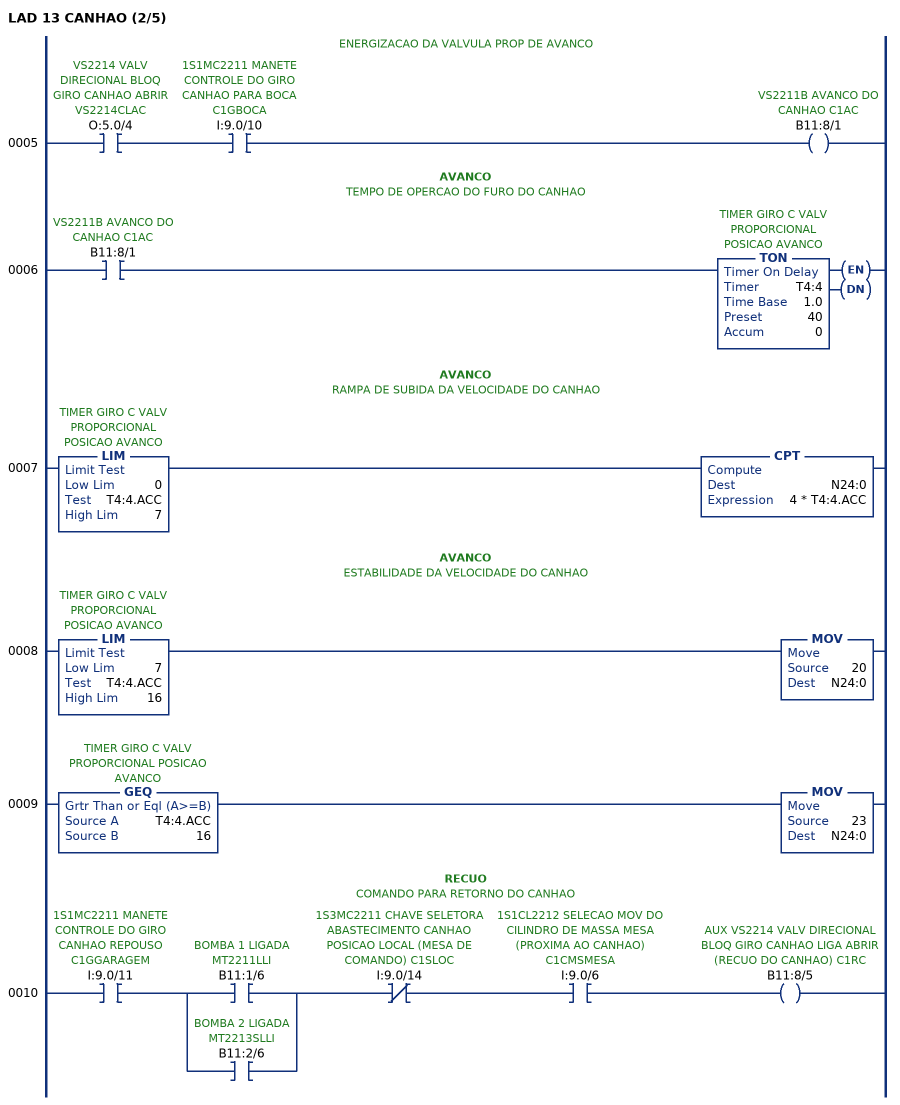
% Rung: 5 %
% ENERGIZACAO DA VALVULA PROP DE AVANCO %
SOR XIC O:5.0/4 XIC I:9.0/10 OTE B11:8/1 EOR
%   O:5.0/4  VS2214CLAC  "VS2214 VALV DIRECIONAL BLOQ GIRO CANHAO ABRIR" %
%   I:9.0/10  C1GBOCA  "1S1MC2211 MANETE CONTROLE DO GIRO CANHAO PARA BOCA" %
%   B11:8/1  C1AC  "VS2211B AVANCO DO CANHAO" %
% Rung: 6 %
% TITLE: AVANCO %
% TEMPO DE OPERCAO DO FURO DO CANHAO %
SOR XIC B11:8/1 TON T4:4 1.0 40 0 EOR
%   B11:8/1  C1AC  "VS2211B AVANCO DO CANHAO" %
%   T4:4  "TIMER GIRO C VALV PROPORCIONAL POSICAO AVANCO" %
% Rung: 7 %
% TITLE: AVANCO %
% RAMPA DE SUBIDA DA VELOCIDADE DO CANHAO %
SOR LIM 0 T4:4.ACC 7 CPT N24:0 " 4 * T4:4.ACC " EOR
%   T4:4  "TIMER GIRO C VALV PROPORCIONAL POSICAO AVANCO" %
% Rung: 8 %
% TITLE: AVANCO %
% ESTABILIDADE DA VELOCIDADE DO CANHAO %
SOR LIM 7 T4:4.ACC 16 MOV 20 N24:0 EOR
%   T4:4  "TIMER GIRO C VALV PROPORCIONAL POSICAO AVANCO" %
% Rung: 9 %
SOR GEQ T4:4.ACC 16 MOV 23 N24:0 EOR
%   T4:4  "TIMER GIRO C VALV PROPORCIONAL POSICAO AVANCO" %
% Rung: 10 %
% TITLE: RECUO %
% COMANDO PARA RETORNO DO CANHAO %
SOR XIC I:9.0/11 BST XIC B11:1/6 NXB XIC B11:2/6 BND XIO I:9.0/14 XIC I:9.0/6 OTE B11:8/5 EOR
%   I:9.0/11  C1GGARAGEM  "1S1MC2211 MANETE CONTROLE DO GIRO CANHAO REPOUSO" %
%   B11:1/6  MT2211LLI  "BOMBA 1 LIGADA" %
%   B11:2/6  MT2213SLLI  "BOMBA 2 LIGADA" %
%   I:9.0/14  C1SLOC  "1S3MC2211 CHAVE SELETORA ABASTECIMENTO CANHAO POSICAO LOCAL (MESA DE COMANDO)" %
%   I:9.0/6  C1CMSMESA  "1S1CL2212 SELECAO MOV DO CILINDRO DE MASSA MESA (PROXIMA AO CANHAO)" %
%   B11:8/5  C1RC  "AUX VS2214 VALV DIRECIONAL BLOQ GIRO CANHAO LIGA ABRIR (RECUO DO CANHAO)" %

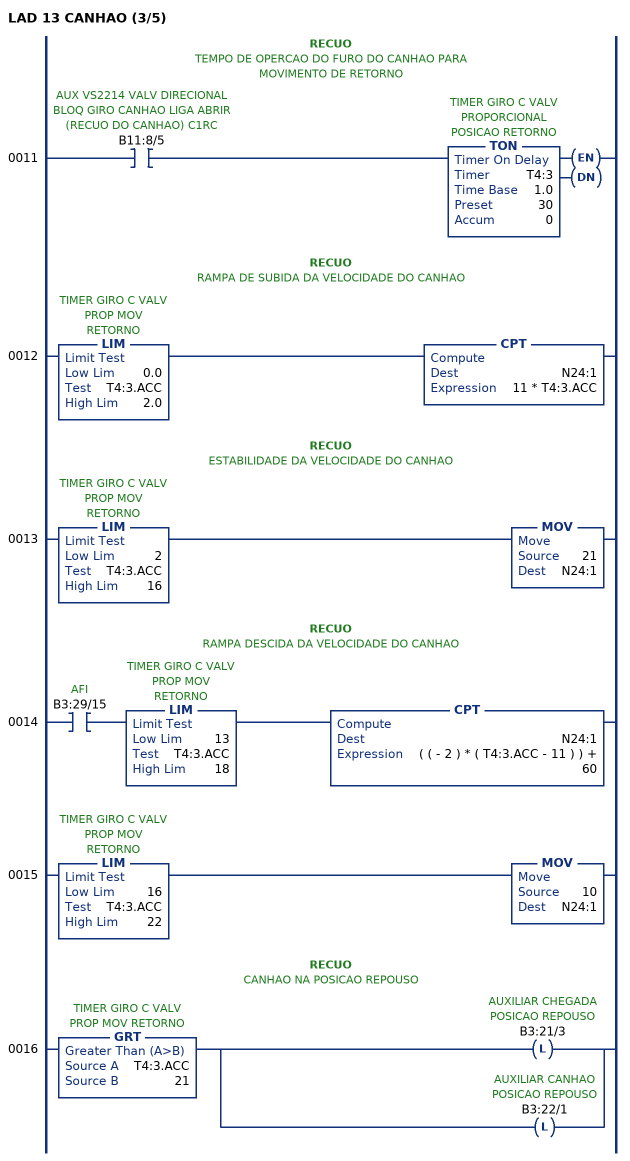
% Rung: 11 %
% TITLE: RECUO %
% TEMPO DE OPERCAO DO FURO DO CANHAO PARA
%  MOVIMENTO DE RETORNO %
SOR XIC B11:8/5 TON T4:3 1.0 30 0 EOR
%   B11:8/5  C1RC  "AUX VS2214 VALV DIRECIONAL BLOQ GIRO CANHAO LIGA ABRIR (RECUO DO CANHAO)" %
%   T4:3  "TIMER GIRO C VALV PROPORCIONAL POSICAO RETORNO" %
% Rung: 12 %
% TITLE: RECUO %
% RAMPA DE SUBIDA DA VELOCIDADE DO CANHAO %
SOR LIM 0.0 T4:3.ACC 2.0 CPT N24:1 " 11 * T4:3.ACC " EOR
%   T4:3.ACC  "TIMER GIRO C VALV PROP MOV RETORNO" %
% Rung: 13 %
% TITLE: RECUO %
% ESTABILIDADE DA VELOCIDADE DO CANHAO %
SOR LIM 2 T4:3.ACC 16 MOV 21 N24:1 EOR
%   T4:3.ACC  "TIMER GIRO C VALV PROP MOV RETORNO" %
% Rung: 14 %
% TITLE: RECUO %
% RAMPA DESCIDA DA VELOCIDADE DO CANHAO %
SOR XIC B3:29/15 LIM 13 T4:3.ACC 18 CPT N24:1 " ( ( - 2 ) * ( T4:3.ACC - 11 ) ) + 60 " EOR
%   B3:29/15  AFI %
%   T4:3.ACC  "TIMER GIRO C VALV PROP MOV RETORNO" %
% Rung: 15 %
SOR LIM 16 T4:3.ACC 22 MOV 10 N24:1 EOR
%   T4:3.ACC  "TIMER GIRO C VALV PROP MOV RETORNO" %
% Rung: 16 %
% TITLE: RECUO %
% CANHAO NA POSICAO REPOUSO %
SOR GRT T4:3.ACC 21 BST OTL B3:21/3 NXB OTL B3:22/1 BND EOR
%   T4:3.ACC  "TIMER GIRO C VALV PROP MOV RETORNO" %
%   B3:21/3  "AUXILIAR CHEGADA POSICAO REPOUSO" %
%   B3:22/1  "AUXILIAR CANHAO POSICAO REPOUSO" %

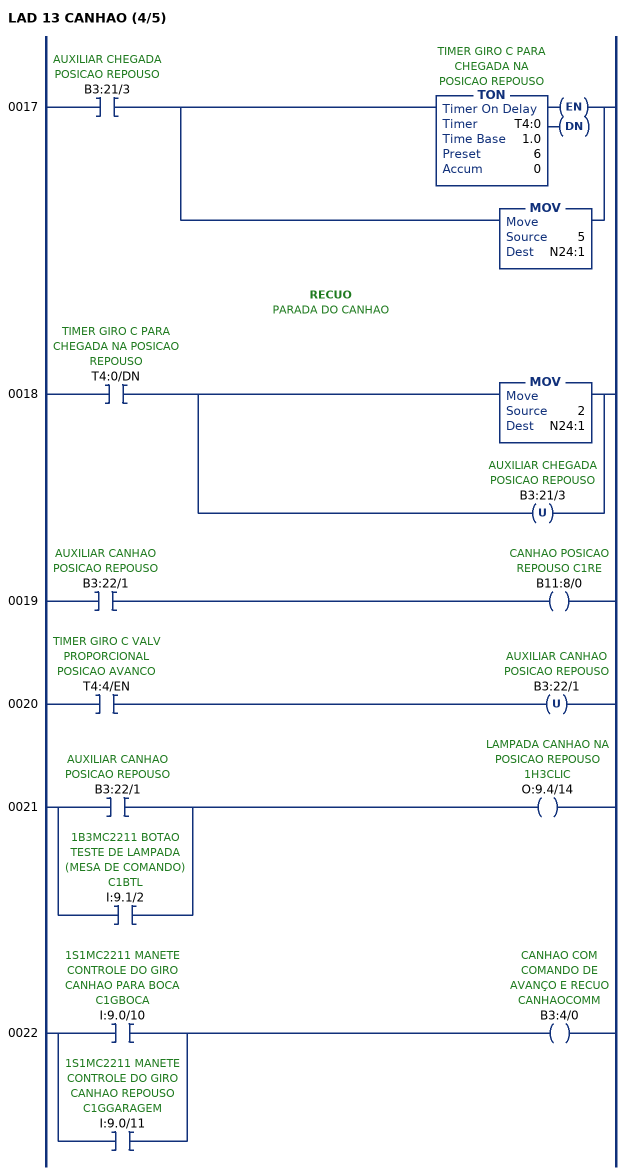
% Rung: 17 %
SOR XIC B3:21/3 BST TON T4:0 1.0 6 0 NXB MOV 5 N24:1 BND EOR
%   B3:21/3  "AUXILIAR CHEGADA POSICAO REPOUSO" %
%   T4:0  "TIMER GIRO C PARA CHEGADA NA POSICAO REPOUSO" %
% Rung: 18 %
% TITLE: RECUO %
% PARADA DO CANHAO %
SOR XIC T4:0/DN BST MOV 2 N24:1 NXB OTU B3:21/3 BND EOR
%   T4:0  "TIMER GIRO C PARA CHEGADA NA POSICAO REPOUSO" %
%   B3:21/3  "AUXILIAR CHEGADA POSICAO REPOUSO" %
% Rung: 19 %
SOR XIC B3:22/1 OTE B11:8/0 EOR
%   B3:22/1  "AUXILIAR CANHAO POSICAO REPOUSO" %
%   B11:8/0  C1RE  "CANHAO POSICAO REPOUSO" %
% Rung: 20 %
SOR XIC T4:4/EN OTU B3:22/1 EOR
%   T4:4  "TIMER GIRO C VALV PROPORCIONAL POSICAO AVANCO" %
%   B3:22/1  "AUXILIAR CANHAO POSICAO REPOUSO" %
% Rung: 21 %
SOR BST XIC B3:22/1 NXB XIC I:9.1/2 BND OTE O:9.4/14 EOR
%   B3:22/1  "AUXILIAR CANHAO POSICAO REPOUSO" %
%   I:9.1/2  C1BTL  "1B3MC2211 BOTAO TESTE DE LAMPADA (MESA DE COMANDO)" %
%   O:9.4/14  1H3CLIC  "LAMPADA CANHAO NA POSICAO REPOUSO" %
% Rung: 22 %
SOR BST XIC I:9.0/10 NXB XIC I:9.0/11 BND OTE B3:4/0 EOR
%   I:9.0/10  C1GBOCA  "1S1MC2211 MANETE CONTROLE DO GIRO CANHAO PARA BOCA" %
%   I:9.0/11  C1GGARAGEM  "1S1MC2211 MANETE CONTROLE DO GIRO CANHAO REPOUSO" %
%   B3:4/0  CANHAOCOMM  "CANHAO COM COMANDO DE AVANÇO E RECUO" %

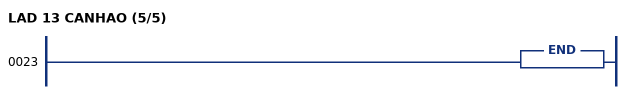
% Rung: 23 %
SOR END EOR

LADDER 14 "INJECAO M"
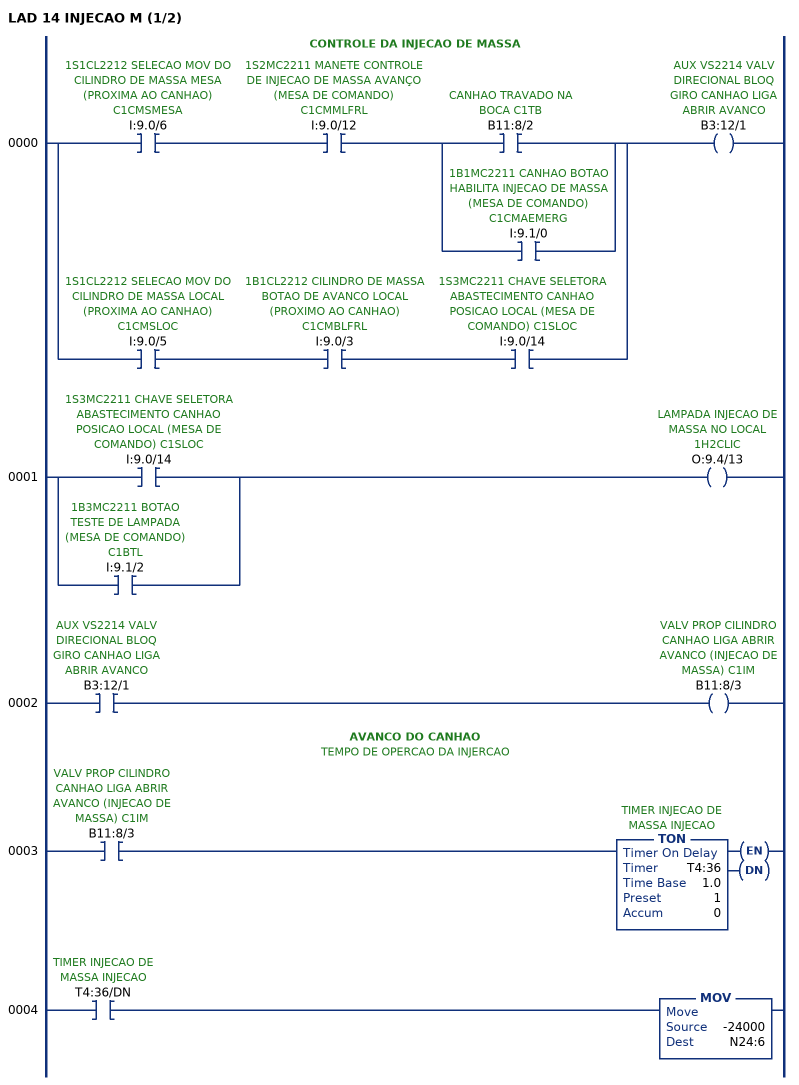
% Rung: 0 %
% TITLE: CONTROLE DA INJECAO DE MASSA %
SOR BST XIC I:9.0/6 XIC I:9.0/12 BST XIC B11:8/2 NXB XIC I:9.1/0 BND NXB XIC I:9.0/5 XIC I:9.0/3 XIC I:9.0/14 BND OTE B3:12/1 EOR
%   I:9.0/6  C1CMSMESA  "1S1CL2212 SELECAO MOV DO CILINDRO DE MASSA MESA (PROXIMA AO CANHAO)" %
%   I:9.0/12  C1CMMLFRL  "1S2MC2211 MANETE CONTROLE DE INJECAO DE MASSA AVANÇO (MESA DE COMANDO)" %
%   B11:8/2  C1TB  "CANHAO TRAVADO NA BOCA" %
%   I:9.1/0  C1CMAEMERG  "1B1MC2211 CANHAO BOTAO HABILITA INJECAO DE MASSA (MESA DE COMANDO)" %
%   I:9.0/5  C1CMSLOC  "1S1CL2212 SELECAO MOV DO CILINDRO DE MASSA LOCAL (PROXIMA AO CANHAO)" %
%   I:9.0/3  C1CMBLFRL  "1B1CL2212 CILINDRO DE MASSA BOTAO DE AVANCO LOCAL (PROXIMO AO CANHAO)" %
%   I:9.0/14  C1SLOC  "1S3MC2211 CHAVE SELETORA ABASTECIMENTO CANHAO POSICAO LOCAL (MESA DE COMANDO)" %
%   B3:12/1  "AUX VS2214 VALV DIRECIONAL BLOQ GIRO CANHAO LIGA ABRIR AVANCO" %
% Rung: 1 %
SOR BST XIC I:9.0/14 NXB XIC I:9.1/2 BND OTE O:9.4/13 EOR
%   I:9.0/14  C1SLOC  "1S3MC2211 CHAVE SELETORA ABASTECIMENTO CANHAO POSICAO LOCAL (MESA DE COMANDO)" %
%   I:9.1/2  C1BTL  "1B3MC2211 BOTAO TESTE DE LAMPADA (MESA DE COMANDO)" %
%   O:9.4/13  1H2CLIC  "LAMPADA INJECAO DE MASSA NO LOCAL" %
% Rung: 2 %
SOR XIC B3:12/1 OTE B11:8/3 EOR
%   B3:12/1  "AUX VS2214 VALV DIRECIONAL BLOQ GIRO CANHAO LIGA ABRIR AVANCO" %
%   B11:8/3  C1IM  "VALV PROP CILINDRO CANHAO LIGA ABRIR AVANCO (INJECAO DE MASSA)" %
% Rung: 3 %
% TITLE: AVANCO DO CANHAO %
% TEMPO DE OPERCAO DA INJERCAO %
SOR XIC B11:8/3 TON T4:36 1.0 1 0 EOR
%   B11:8/3  C1IM  "VALV PROP CILINDRO CANHAO LIGA ABRIR AVANCO (INJECAO DE MASSA)" %
%   T4:36  "TIMER INJECAO DE MASSA INJECAO" %
% Rung: 4 %
SOR XIC T4:36/DN MOV -24000 N24:6 EOR
%   T4:36  "TIMER INJECAO DE MASSA INJECAO" %

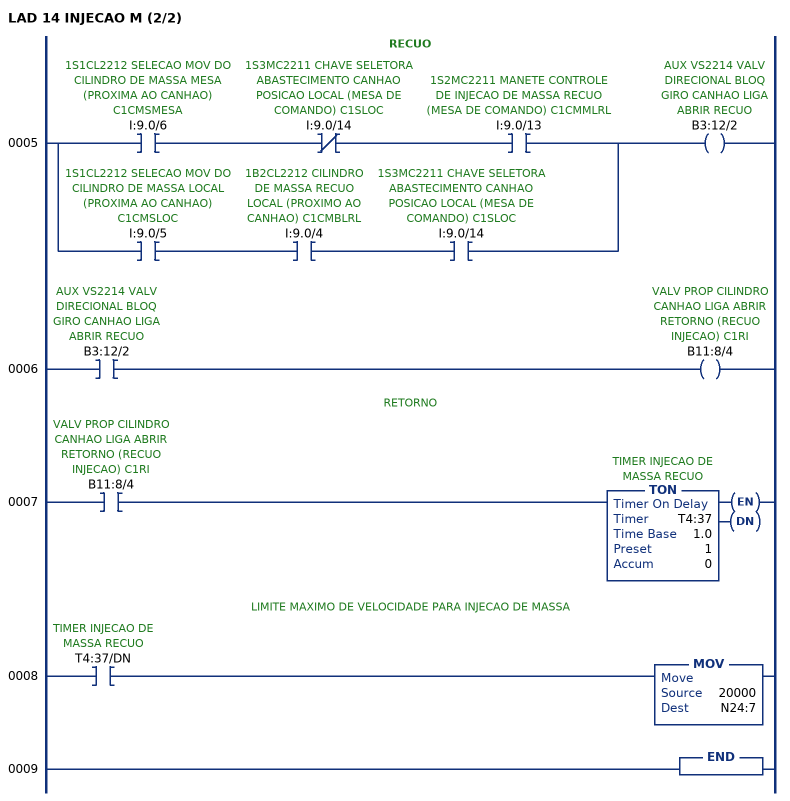
% Rung: 5 %
% TITLE: RECUO %
SOR BST XIC I:9.0/6 XIO I:9.0/14 XIC I:9.0/13 NXB XIC I:9.0/5 XIC I:9.0/4 XIC I:9.0/14 BND OTE B3:12/2 EOR
%   I:9.0/6  C1CMSMESA  "1S1CL2212 SELECAO MOV DO CILINDRO DE MASSA MESA (PROXIMA AO CANHAO)" %
%   I:9.0/14  C1SLOC  "1S3MC2211 CHAVE SELETORA ABASTECIMENTO CANHAO POSICAO LOCAL (MESA DE COMANDO)" %
%   I:9.0/13  C1CMMLRL  "1S2MC2211 MANETE CONTROLE DE INJECAO DE MASSA RECUO (MESA DE COMANDO)" %
%   I:9.0/5  C1CMSLOC  "1S1CL2212 SELECAO MOV DO CILINDRO DE MASSA LOCAL (PROXIMA AO CANHAO)" %
%   I:9.0/4  C1CMBLRL  "1B2CL2212 CILINDRO DE MASSA RECUO LOCAL (PROXIMO AO CANHAO)" %
%   B3:12/2  "AUX VS2214 VALV DIRECIONAL BLOQ GIRO CANHAO LIGA ABRIR RECUO" %
% Rung: 6 %
SOR XIC B3:12/2 OTE B11:8/4 EOR
%   B3:12/2  "AUX VS2214 VALV DIRECIONAL BLOQ GIRO CANHAO LIGA ABRIR RECUO" %
%   B11:8/4  C1RI  "VALV PROP CILINDRO CANHAO LIGA ABRIR RETORNO (RECUO INJECAO)" %
% Rung: 7 %
% RETORNO %
SOR XIC B11:8/4 TON T4:37 1.0 1 0 EOR
%   B11:8/4  C1RI  "VALV PROP CILINDRO CANHAO LIGA ABRIR RETORNO (RECUO INJECAO)" %
%   T4:37  "TIMER INJECAO DE MASSA RECUO" %
% Rung: 8 %
% LIMITE MAXIMO DE VELOCIDADE PARA INJECAO DE MASSA %
SOR XIC T4:37/DN MOV 20000 N24:7 EOR
%   T4:37  "TIMER INJECAO DE MASSA RECUO" %
% Rung: 9 %
SOR END EOR

LADDER 15 "PERFURAT"
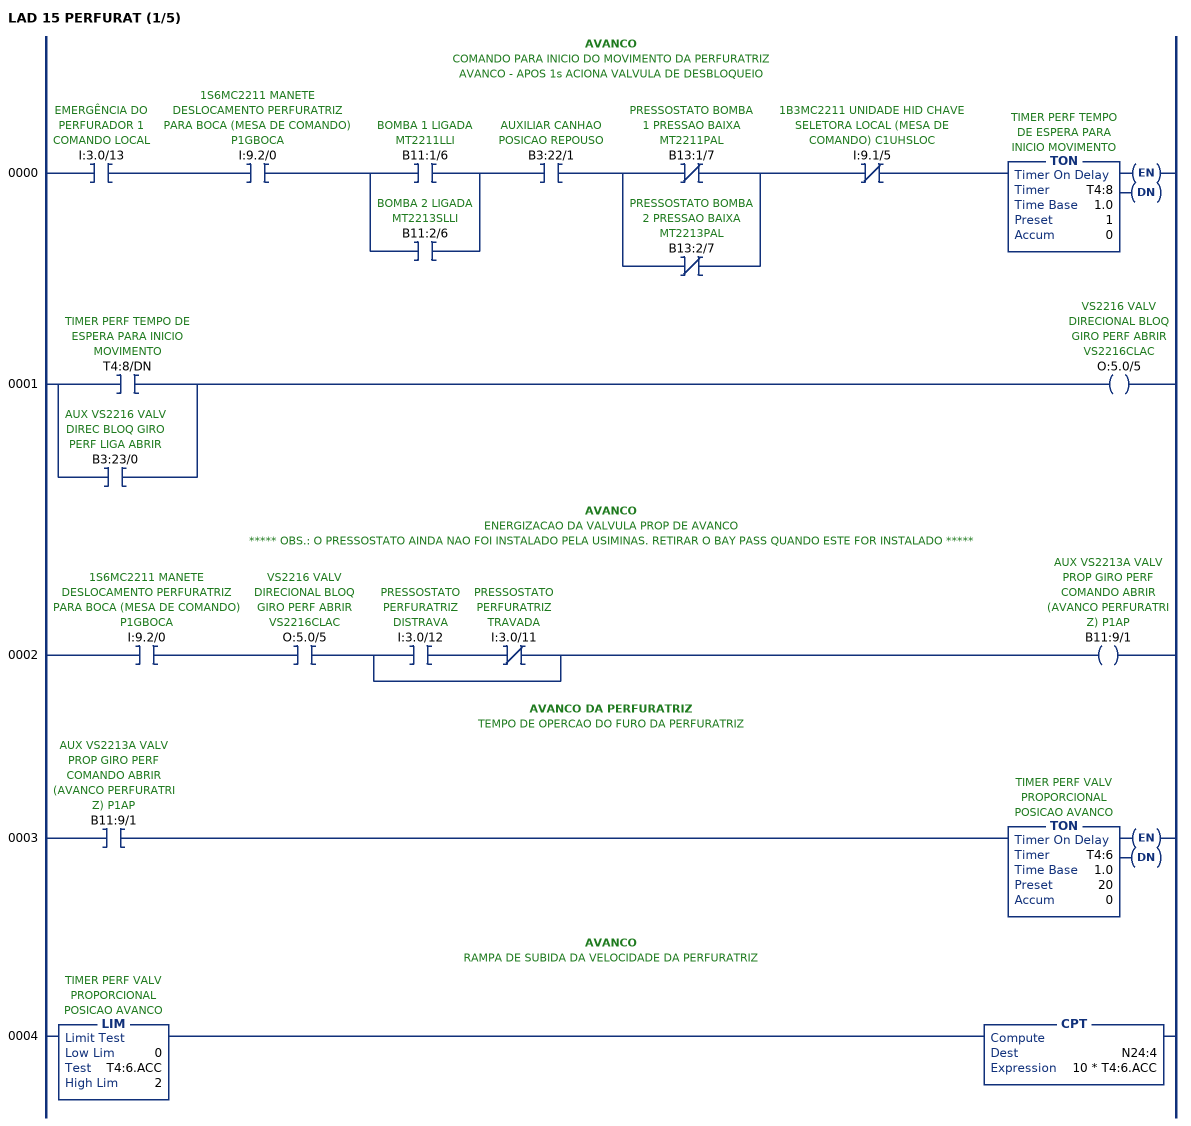
% Rung: 0 %
% TITLE: AVANCO %
% COMANDO PARA INICIO DO MOVIMENTO DA PERFURATRIZ
% AVANCO - APOS 1s ACIONA VALVULA DE DESBLOQUEIO %
SOR XIC I:3.0/13 XIC I:9.2/0 BST XIC B11:1/6 NXB XIC B11:2/6 BND XIC B3:22/1 BST XIO B13:1/7 NXB XIO B13:2/7 BND XIO I:9.1/5 TON T4:8 1.0 1 0 EOR
%   I:3.0/13  "EMERGÊNCIA DO PERFURADOR 1 COMANDO LOCAL" %
%   I:9.2/0  P1GBOCA  "1S6MC2211 MANETE DESLOCAMENTO PERFURATRIZ PARA BOCA (MESA DE COMANDO)" %
%   B11:1/6  MT2211LLI  "BOMBA 1 LIGADA" %
%   B11:2/6  MT2213SLLI  "BOMBA 2 LIGADA" %
%   B3:22/1  "AUXILIAR CANHAO POSICAO REPOUSO" %
%   B13:1/7  MT2211PAL  "PRESSOSTATO BOMBA 1 PRESSAO BAIXA" %
%   B13:2/7  MT2213PAL  "PRESSOSTATO BOMBA 2 PRESSAO BAIXA" %
%   I:9.1/5  C1UHSLOC  "1B3MC2211 UNIDADE HID CHAVE SELETORA LOCAL (MESA DE COMANDO)" %
%   T4:8  "TIMER PERF TEMPO DE ESPERA PARA INICIO MOVIMENTO" %
% Rung: 1 %
SOR BST XIC T4:8/DN NXB XIC B3:23/0 BND OTE O:5.0/5 EOR
%   T4:8  "TIMER PERF TEMPO DE ESPERA PARA INICIO MOVIMENTO" %
%   B3:23/0  "AUX VS2216 VALV DIREC BLOQ GIRO PERF LIGA ABRIR" %
%   O:5.0/5  VS2216CLAC  "VS2216 VALV DIRECIONAL BLOQ GIRO PERF ABRIR" %
% Rung: 2 %
% TITLE: AVANCO %
% ENERGIZACAO DA VALVULA PROP DE AVANCO
% ***** OBS.: O PRESSOSTATO AINDA NAO FOI INSTALADO PELA USIMINAS. RETIRAR O BAY PASS QUANDO ESTE FOR INSTALADO ***** %
SOR XIC I:9.2/0 XIC O:5.0/5 BST XIC I:3.0/12 XIO I:3.0/11 NXB BND OTE B11:9/1 EOR
%   I:9.2/0  P1GBOCA  "1S6MC2211 MANETE DESLOCAMENTO PERFURATRIZ PARA BOCA (MESA DE COMANDO)" %
%   O:5.0/5  VS2216CLAC  "VS2216 VALV DIRECIONAL BLOQ GIRO PERF ABRIR" %
%   I:3.0/12  "PRESSOSTATO PERFURATRIZ DISTRAVA" %
%   I:3.0/11  "PRESSOSTATO PERFURATRIZ TRAVADA" %
%   B11:9/1  P1AP  "AUX VS2213A VALV PROP GIRO PERF COMANDO ABRIR (AVANCO PERFURATRIZ)" %
% Rung: 3 %
% TITLE: AVANCO DA PERFURATRIZ %
% TEMPO DE OPERCAO DO FURO DA PERFURATRIZ %
SOR XIC B11:9/1 TON T4:6 1.0 20 0 EOR
%   B11:9/1  P1AP  "AUX VS2213A VALV PROP GIRO PERF COMANDO ABRIR (AVANCO PERFURATRIZ)" %
%   T4:6  "TIMER PERF VALV PROPORCIONAL POSICAO AVANCO" %
% Rung: 4 %
% TITLE: AVANCO %
% RAMPA DE SUBIDA DA VELOCIDADE DA PERFURATRIZ %
SOR LIM 0 T4:6.ACC 2 CPT N24:4 " 10 * T4:6.ACC " EOR
%   T4:6  "TIMER PERF VALV PROPORCIONAL POSICAO AVANCO" %

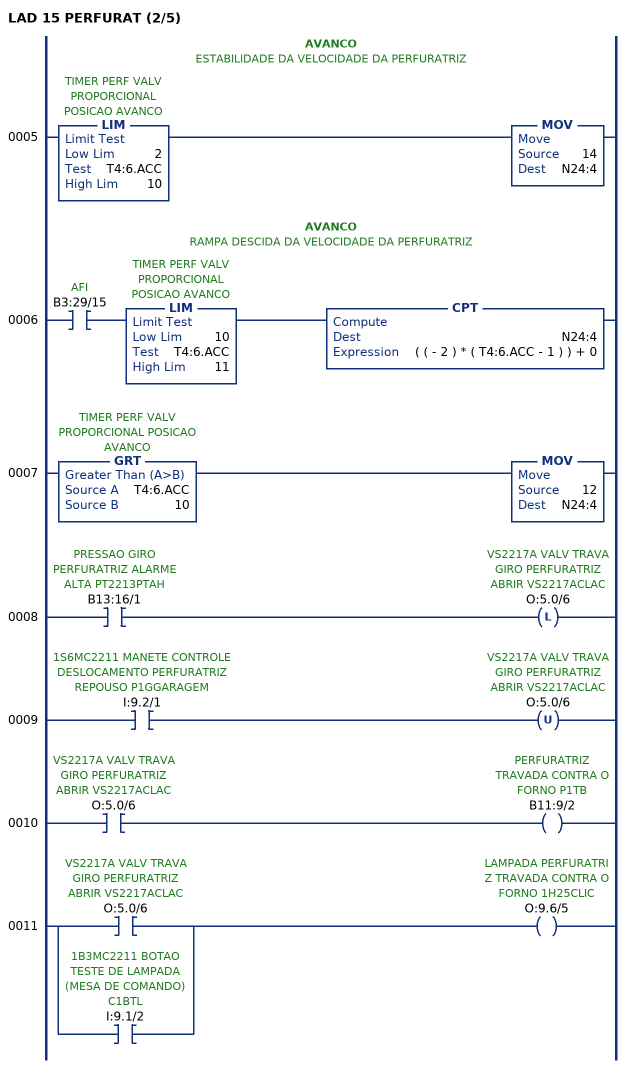
% Rung: 5 %
% TITLE: AVANCO %
% ESTABILIDADE DA VELOCIDADE DA PERFURATRIZ %
SOR LIM 2 T4:6.ACC 10 MOV 14 N24:4 EOR
%   T4:6  "TIMER PERF VALV PROPORCIONAL POSICAO AVANCO" %
% Rung: 6 %
% TITLE: AVANCO %
% RAMPA DESCIDA DA VELOCIDADE DA PERFURATRIZ %
SOR XIC B3:29/15 LIM 10 T4:6.ACC 11 CPT N24:4 " ( ( - 2 ) * ( T4:6.ACC - 1 ) ) + 0 " EOR
%   B3:29/15  AFI %
%   T4:6  "TIMER PERF VALV PROPORCIONAL POSICAO AVANCO" %
% Rung: 7 %
SOR GRT T4:6.ACC 10 MOV 12 N24:4 EOR
%   T4:6  "TIMER PERF VALV PROPORCIONAL POSICAO AVANCO" %
% Rung: 8 %
SOR XIC B13:16/1 OTL O:5.0/6 EOR
%   B13:16/1  PT2213PTAH  "PRESSAO GIRO PERFURATRIZ ALARME ALTA" %
%   O:5.0/6  VS2217ACLAC  "VS2217A VALV TRAVA GIRO PERFURATRIZ ABRIR" %
% Rung: 9 %
SOR XIC I:9.2/1 OTU O:5.0/6 EOR
%   I:9.2/1  P1GGARAGEM  "1S6MC2211 MANETE CONTROLE DESLOCAMENTO PERFURATRIZ REPOUSO" %
%   O:5.0/6  VS2217ACLAC  "VS2217A VALV TRAVA GIRO PERFURATRIZ ABRIR" %
% Rung: 10 %
SOR XIC O:5.0/6 OTE B11:9/2 EOR
%   O:5.0/6  VS2217ACLAC  "VS2217A VALV TRAVA GIRO PERFURATRIZ ABRIR" %
%   B11:9/2  P1TB  "PERFURATRIZ TRAVADA CONTRA O FORNO" %
% Rung: 11 %
SOR BST XIC O:5.0/6 NXB XIC I:9.1/2 BND OTE O:9.6/5 EOR
%   O:5.0/6  VS2217ACLAC  "VS2217A VALV TRAVA GIRO PERFURATRIZ ABRIR" %
%   I:9.1/2  C1BTL  "1B3MC2211 BOTAO TESTE DE LAMPADA (MESA DE COMANDO)" %
%   O:9.6/5  1H25CLIC  "LAMPADA PERFURATRIZ TRAVADA CONTRA O FORNO" %

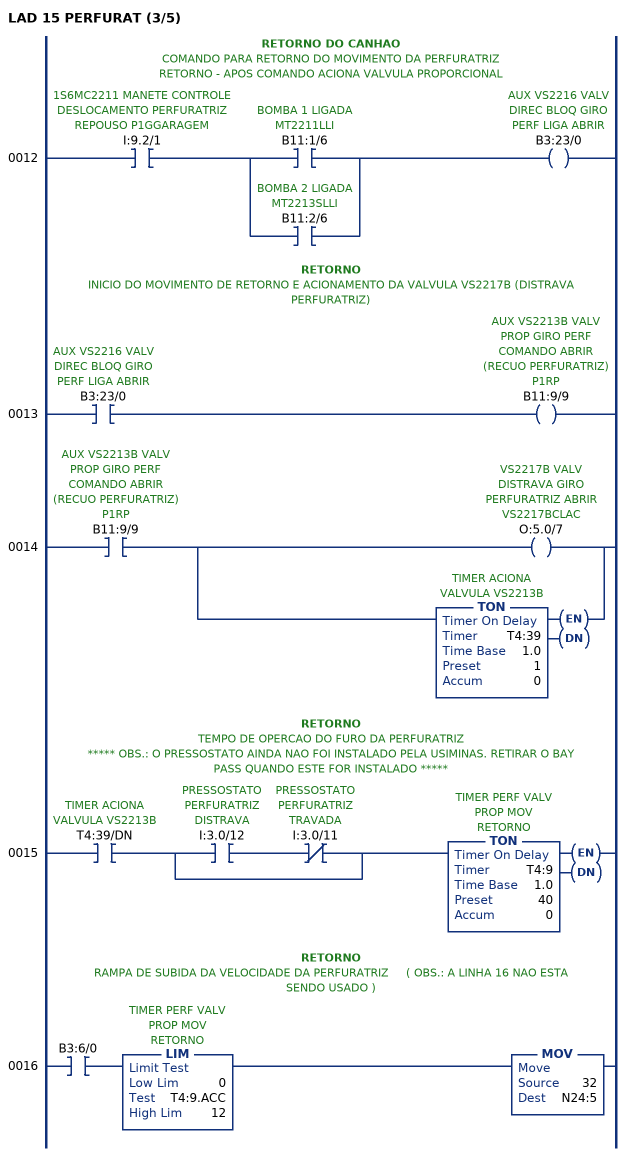
% Rung: 12 %
% TITLE: RETORNO DO CANHAO %
% COMANDO PARA RETORNO DO MOVIMENTO DA PERFURATRIZ
% RETORNO - APOS COMANDO ACIONA VALVULA PROPORCIONAL %
SOR XIC I:9.2/1 BST XIC B11:1/6 NXB XIC B11:2/6 BND OTE B3:23/0 EOR
%   I:9.2/1  P1GGARAGEM  "1S6MC2211 MANETE CONTROLE DESLOCAMENTO PERFURATRIZ REPOUSO" %
%   B11:1/6  MT2211LLI  "BOMBA 1 LIGADA" %
%   B11:2/6  MT2213SLLI  "BOMBA 2 LIGADA" %
%   B3:23/0  "AUX VS2216 VALV DIREC BLOQ GIRO PERF LIGA ABRIR" %
% Rung: 13 %
% TITLE: RETORNO %
% INICIO DO MOVIMENTO DE RETORNO E ACIONAMENTO DA VALVULA VS2217B (DISTRAVA PERFURATRIZ) %
SOR XIC B3:23/0 OTE B11:9/9 EOR
%   B3:23/0  "AUX VS2216 VALV DIREC BLOQ GIRO PERF LIGA ABRIR" %
%   B11:9/9  P1RP  "AUX VS2213B VALV PROP GIRO PERF COMANDO ABRIR (RECUO PERFURATRIZ)" %
% Rung: 14 %
SOR XIC B11:9/9 BST OTE O:5.0/7 NXB TON T4:39 1.0 1 0 BND EOR
%   B11:9/9  P1RP  "AUX VS2213B VALV PROP GIRO PERF COMANDO ABRIR (RECUO PERFURATRIZ)" %
%   O:5.0/7  VS2217BCLAC  "VS2217B VALV DISTRAVA GIRO PERFURATRIZ ABRIR" %
%   T4:39  "TIMER ACIONA VALVULA VS2213B" %
% Rung: 15 %
% TITLE: RETORNO %
% TEMPO DE OPERCAO DO FURO DA PERFURATRIZ
% ***** OBS.: O PRESSOSTATO AINDA NAO FOI INSTALADO PELA USIMINAS. RETIRAR O BAY PASS QUANDO ESTE FOR INSTALADO ***** %
SOR XIC T4:39/DN BST XIC I:3.0/12 XIO I:3.0/11 NXB BND TON T4:9 1.0 40 0 EOR
%   T4:39  "TIMER ACIONA VALVULA VS2213B" %
%   I:3.0/12  "PRESSOSTATO PERFURATRIZ DISTRAVA" %
%   I:3.0/11  "PRESSOSTATO PERFURATRIZ TRAVADA" %
%   T4:9  "TIMER PERF VALV PROP MOV RETORNO" %
% Rung: 16 %
% TITLE: RETORNO %
% RAMPA DE SUBIDA DA VELOCIDADE DA PERFURATRIZ     ( OBS.: A LINHA 16 NAO ESTA SENDO USADO ) %
SOR XIC B3:6/0 LIM 0 T4:9.ACC 12 MOV 32 N24:5 EOR
%   T4:9  "TIMER PERF VALV PROP MOV RETORNO" %

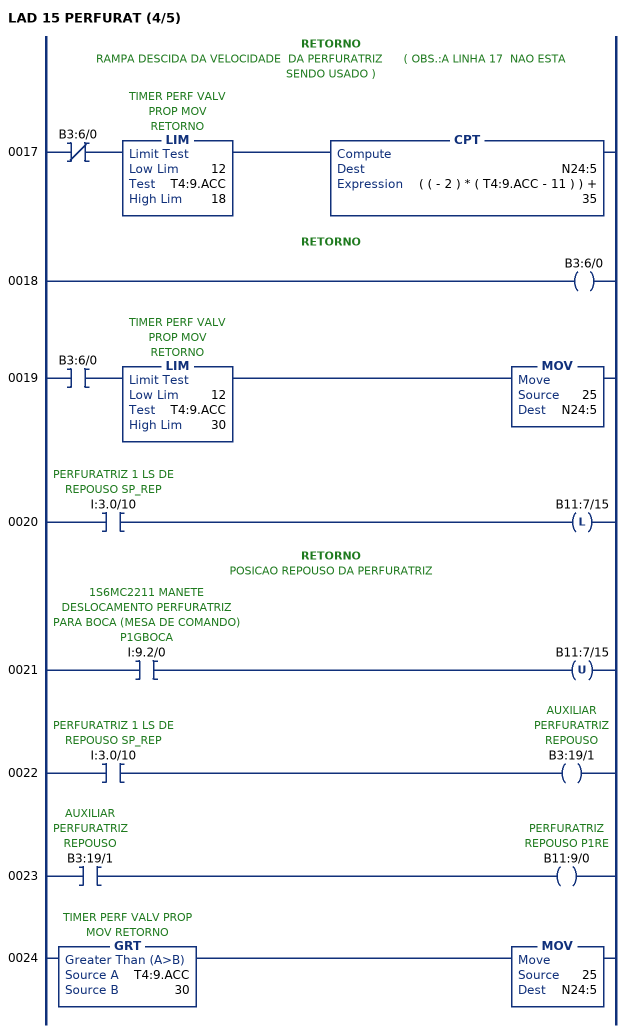
% Rung: 17 %
% TITLE: RETORNO %
% RAMPA DESCIDA DA VELOCIDADE  DA PERFURATRIZ      ( OBS.:A LINHA 17  NAO ESTA SENDO USADO ) %
SOR XIO B3:6/0 LIM 12 T4:9.ACC 18 CPT N24:5 " ( ( - 2 ) * ( T4:9.ACC - 11 ) ) + 35 " EOR
%   T4:9  "TIMER PERF VALV PROP MOV RETORNO" %
% Rung: 18 %
% TITLE: RETORNO %
SOR OTE B3:6/0 EOR
% Rung: 19 %
SOR XIC B3:6/0 LIM 12 T4:9.ACC 30 MOV 25 N24:5 EOR
%   T4:9  "TIMER PERF VALV PROP MOV RETORNO" %
% Rung: 20 %
SOR XIC I:3.0/10 OTL B11:7/15 EOR
%   I:3.0/10  SP_REP  "PERFURATRIZ 1 LS DE REPOUSO" %
% Rung: 21 %
% TITLE: RETORNO %
% POSICAO REPOUSO DA PERFURATRIZ %
SOR XIC I:9.2/0 OTU B11:7/15 EOR
%   I:9.2/0  P1GBOCA  "1S6MC2211 MANETE DESLOCAMENTO PERFURATRIZ PARA BOCA (MESA DE COMANDO)" %
% Rung: 22 %
SOR XIC I:3.0/10 OTE B3:19/1 EOR
%   I:3.0/10  SP_REP  "PERFURATRIZ 1 LS DE REPOUSO" %
%   B3:19/1  "AUXILIAR PERFURATRIZ REPOUSO" %
% Rung: 23 %
SOR XIC B3:19/1 OTE B11:9/0 EOR
%   B3:19/1  "AUXILIAR PERFURATRIZ REPOUSO" %
%   B11:9/0  P1RE  "PERFURATRIZ REPOUSO" %
% Rung: 24 %
SOR GRT T4:9.ACC 30 MOV 25 N24:5 EOR
%   T4:9  "TIMER PERF VALV PROP MOV RETORNO" %

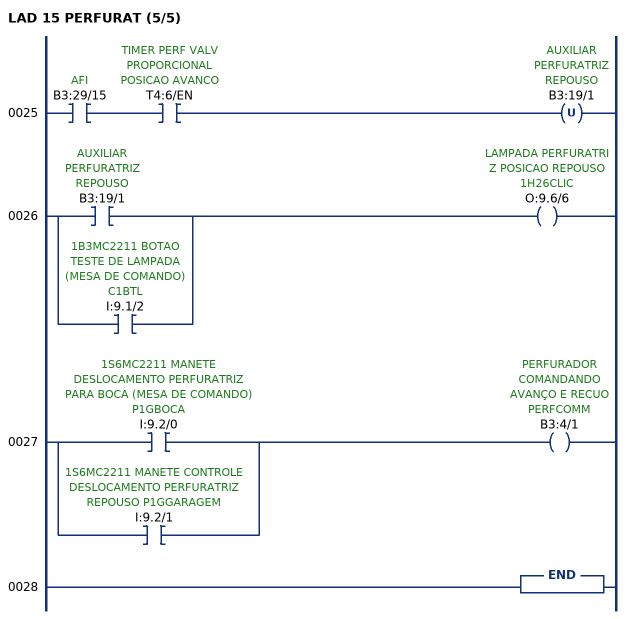
% Rung: 25 %
SOR XIC B3:29/15 XIC T4:6/EN OTU B3:19/1 EOR
%   B3:29/15  AFI %
%   T4:6  "TIMER PERF VALV PROPORCIONAL POSICAO AVANCO" %
%   B3:19/1  "AUXILIAR PERFURATRIZ REPOUSO" %
% Rung: 26 %
SOR BST XIC B3:19/1 NXB XIC I:9.1/2 BND OTE O:9.6/6 EOR
%   B3:19/1  "AUXILIAR PERFURATRIZ REPOUSO" %
%   I:9.1/2  C1BTL  "1B3MC2211 BOTAO TESTE DE LAMPADA (MESA DE COMANDO)" %
%   O:9.6/6  1H26CLIC  "LAMPADA PERFURATRIZ POSICAO REPOUSO" %
% Rung: 27 %
SOR BST XIC I:9.2/0 NXB XIC I:9.2/1 BND OTE B3:4/1 EOR
%   I:9.2/0  P1GBOCA  "1S6MC2211 MANETE DESLOCAMENTO PERFURATRIZ PARA BOCA (MESA DE COMANDO)" %
%   I:9.2/1  P1GGARAGEM  "1S6MC2211 MANETE CONTROLE DESLOCAMENTO PERFURATRIZ REPOUSO" %
%   B3:4/1  PERFCOMM  "PERFURADOR COMANDANDO AVANÇO E RECUO" %
% Rung: 28 %
SOR END EOR

LADDER 16 "MARTELETE"
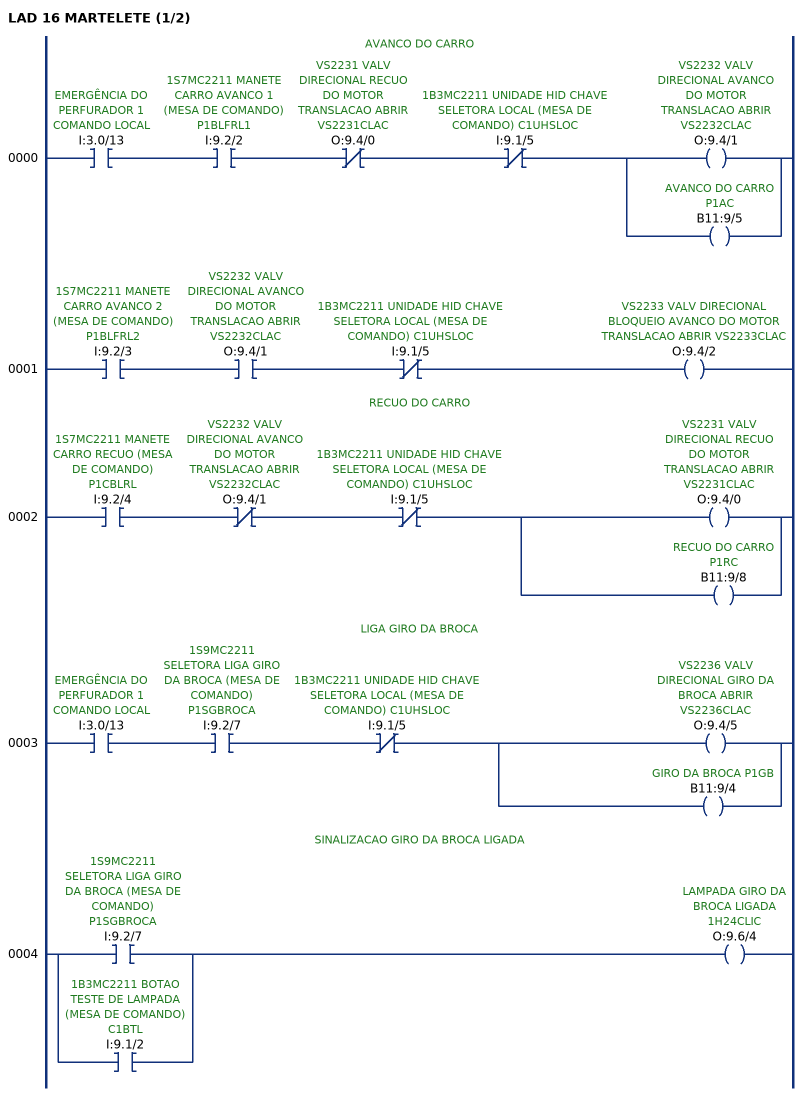
% Rung: 0 %
% AVANCO DO CARRO %
SOR XIC I:3.0/13 XIC I:9.2/2 XIO O:9.4/0 XIO I:9.1/5 BST OTE O:9.4/1 NXB OTE B11:9/5 BND EOR
%   I:3.0/13  "EMERGÊNCIA DO PERFURADOR 1 COMANDO LOCAL" %
%   I:9.2/2  P1BLFRL1  "1S7MC2211 MANETE CARRO AVANCO 1 (MESA DE COMANDO)" %
%   O:9.4/0  VS2231CLAC  "VS2231 VALV DIRECIONAL RECUO DO MOTOR TRANSLACAO ABRIR" %
%   I:9.1/5  C1UHSLOC  "1B3MC2211 UNIDADE HID CHAVE SELETORA LOCAL (MESA DE COMANDO)" %
%   O:9.4/1  VS2232CLAC  "VS2232 VALV DIRECIONAL AVANCO DO MOTOR TRANSLACAO ABRIR" %
%   B11:9/5  P1AC  "AVANCO DO CARRO" %
% Rung: 1 %
SOR XIC I:9.2/3 XIC O:9.4/1 XIO I:9.1/5 OTE O:9.4/2 EOR
%   I:9.2/3  P1BLFRL2  "1S7MC2211 MANETE CARRO AVANCO 2 (MESA DE COMANDO)" %
%   O:9.4/1  VS2232CLAC  "VS2232 VALV DIRECIONAL AVANCO DO MOTOR TRANSLACAO ABRIR" %
%   I:9.1/5  C1UHSLOC  "1B3MC2211 UNIDADE HID CHAVE SELETORA LOCAL (MESA DE COMANDO)" %
%   O:9.4/2  VS2233CLAC  "VS2233 VALV DIRECIONAL BLOQUEIO AVANCO DO MOTOR TRANSLACAO ABRIR" %
% Rung: 2 %
% RECUO DO CARRO %
SOR XIC I:9.2/4 XIO O:9.4/1 XIO I:9.1/5 BST OTE O:9.4/0 NXB OTE B11:9/8 BND EOR
%   I:9.2/4  P1CBLRL  "1S7MC2211 MANETE CARRO RECUO (MESA DE COMANDO)" %
%   O:9.4/1  VS2232CLAC  "VS2232 VALV DIRECIONAL AVANCO DO MOTOR TRANSLACAO ABRIR" %
%   I:9.1/5  C1UHSLOC  "1B3MC2211 UNIDADE HID CHAVE SELETORA LOCAL (MESA DE COMANDO)" %
%   O:9.4/0  VS2231CLAC  "VS2231 VALV DIRECIONAL RECUO DO MOTOR TRANSLACAO ABRIR" %
%   B11:9/8  P1RC  "RECUO DO CARRO" %
% Rung: 3 %
% LIGA GIRO DA BROCA %
SOR XIC I:3.0/13 XIC I:9.2/7 XIO I:9.1/5 BST OTE O:9.4/5 NXB OTE B11:9/4 BND EOR
%   I:3.0/13  "EMERGÊNCIA DO PERFURADOR 1 COMANDO LOCAL" %
%   I:9.2/7  P1SGBROCA  "1S9MC2211 SELETORA LIGA GIRO DA BROCA (MESA DE COMANDO)" %
%   I:9.1/5  C1UHSLOC  "1B3MC2211 UNIDADE HID CHAVE SELETORA LOCAL (MESA DE COMANDO)" %
%   O:9.4/5  VS2236CLAC  "VS2236 VALV DIRECIONAL GIRO DA BROCA ABRIR" %
%   B11:9/4  P1GB  "GIRO DA BROCA" %
% Rung: 4 %
% SINALIZACAO GIRO DA BROCA LIGADA %
SOR BST XIC I:9.2/7 NXB XIC I:9.1/2 BND OTE O:9.6/4 EOR
%   I:9.2/7  P1SGBROCA  "1S9MC2211 SELETORA LIGA GIRO DA BROCA (MESA DE COMANDO)" %
%   I:9.1/2  C1BTL  "1B3MC2211 BOTAO TESTE DE LAMPADA (MESA DE COMANDO)" %
%   O:9.6/4  1H24CLIC  "LAMPADA GIRO DA BROCA LIGADA" %

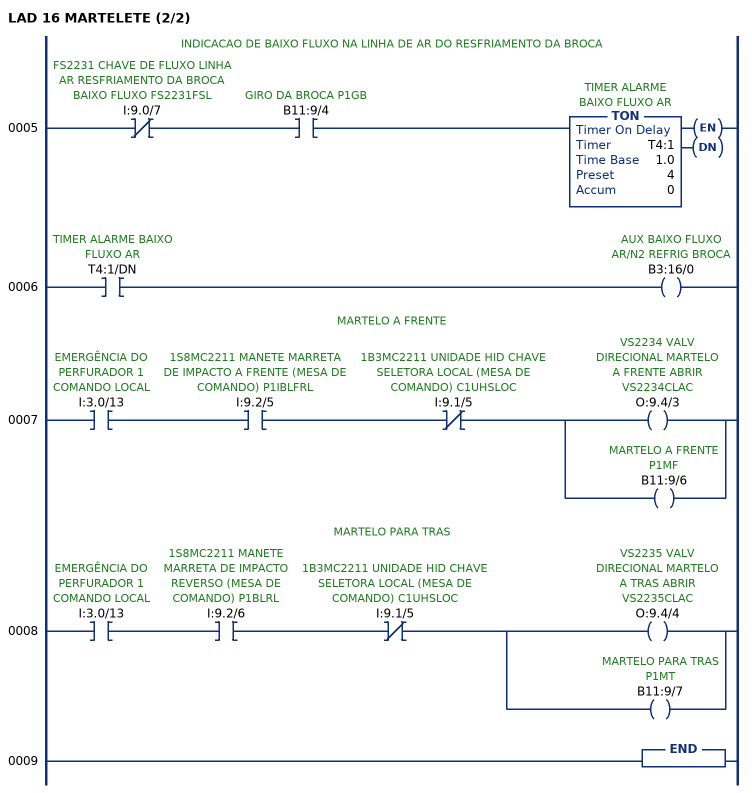
% Rung: 5 %
% INDICACAO DE BAIXO FLUXO NA LINHA DE AR DO RESFRIAMENTO DA BROCA %
SOR XIO I:9.0/7 XIC B11:9/4 TON T4:1 1.0 4 0 EOR
%   I:9.0/7  FS2231FSL  "FS2231 CHAVE DE FLUXO LINHA AR RESFRIAMENTO DA BROCA BAIXO FLUXO" %
%   B11:9/4  P1GB  "GIRO DA BROCA" %
%   T4:1  "TIMER ALARME BAIXO FLUXO AR" %
% Rung: 6 %
SOR XIC T4:1/DN OTE B3:16/0 EOR
%   T4:1  "TIMER ALARME BAIXO FLUXO AR" %
%   B3:16/0  "AUX BAIXO FLUXO AR/N2 REFRIG BROCA" %
% Rung: 7 %
% MARTELO A FRENTE %
SOR XIC I:3.0/13 XIC I:9.2/5 XIO I:9.1/5 BST OTE O:9.4/3 NXB OTE B11:9/6 BND EOR
%   I:3.0/13  "EMERGÊNCIA DO PERFURADOR 1 COMANDO LOCAL" %
%   I:9.2/5  P1IBLFRL  "1S8MC2211 MANETE MARRETA DE IMPACTO A FRENTE (MESA DE COMANDO)" %
%   I:9.1/5  C1UHSLOC  "1B3MC2211 UNIDADE HID CHAVE SELETORA LOCAL (MESA DE COMANDO)" %
%   O:9.4/3  VS2234CLAC  "VS2234 VALV DIRECIONAL MARTELO A FRENTE ABRIR" %
%   B11:9/6  P1MF  "MARTELO A FRENTE" %
% Rung: 8 %
% MARTELO PARA TRAS %
SOR XIC I:3.0/13 XIC I:9.2/6 XIO I:9.1/5 BST OTE O:9.4/4 NXB OTE B11:9/7 BND EOR
%   I:3.0/13  "EMERGÊNCIA DO PERFURADOR 1 COMANDO LOCAL" %
%   I:9.2/6  P1BLRL  "1S8MC2211 MANETE MARRETA DE IMPACTO REVERSO (MESA DE COMANDO)" %
%   I:9.1/5  C1UHSLOC  "1B3MC2211 UNIDADE HID CHAVE SELETORA LOCAL (MESA DE COMANDO)" %
%   O:9.4/4  VS2235CLAC  "VS2235 VALV DIRECIONAL MARTELO A TRAS ABRIR" %
%   B11:9/7  P1MT  "MARTELO PARA TRAS" %
% Rung: 9 %
SOR END EOR

LADDER 17 "BOMBA AGUA"    % Resfriamento da Broca ou Sopro %
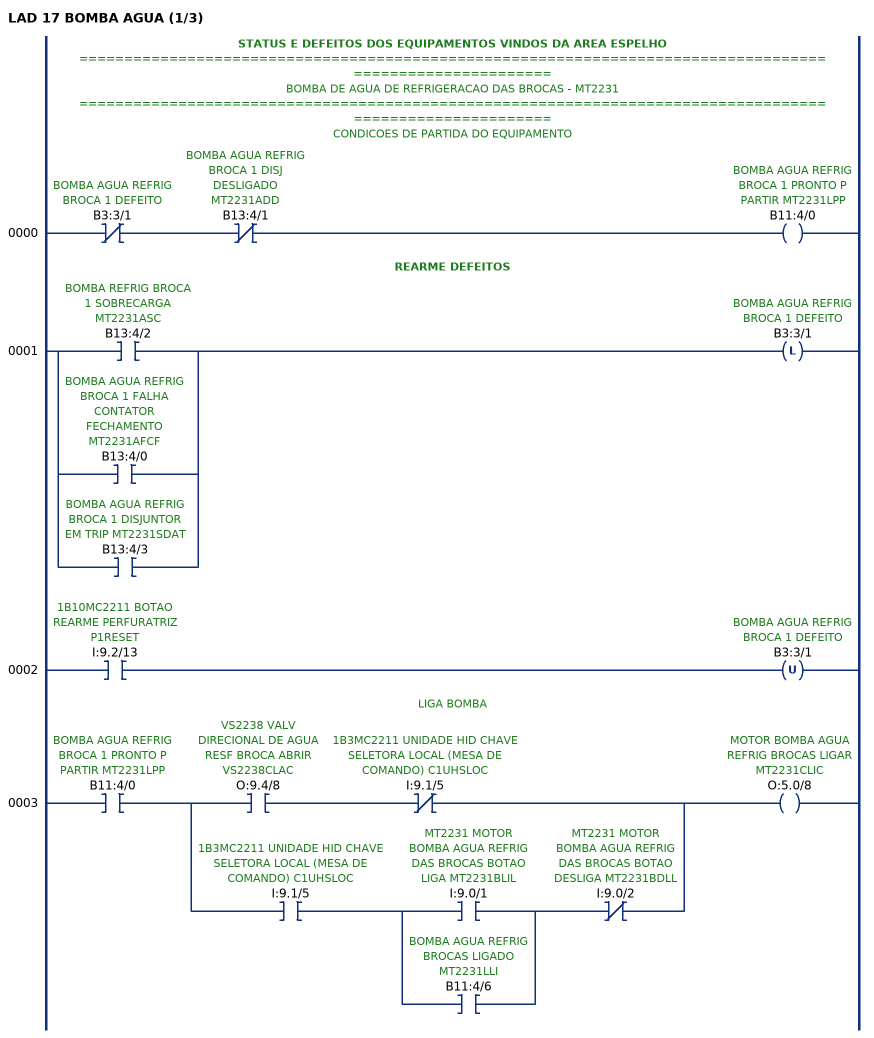
% Rung: 0 %
% TITLE: STATUS E DEFEITOS DOS EQUIPAMENTOS VINDOS DA AREA ESPELHO %
% =========================================================================================================
% BOMBA DE AGUA DE REFRIGERACAO DAS BROCAS - MT2231
% =========================================================================================================
% CONDICOES DE PARTIDA DO EQUIPAMENTO %
SOR XIO B3:3/1 XIO B13:4/1 OTE B11:4/0 EOR
%   B3:3/1  "BOMBA AGUA REFRIG BROCA 1 DEFEITO" %
%   B13:4/1  MT2231ADD  "BOMBA AGUA REFRIG BROCA 1 DISJ DESLIGADO" %
%   B11:4/0  MT2231LPP  "BOMBA AGUA REFRIG BROCA 1 PRONTO P PARTIR" %
% Rung: 1 %
% TITLE: REARME DEFEITOS %
SOR BST XIC B13:4/2 NXB XIC B13:4/0 NXB XIC B13:4/3 BND OTL B3:3/1 EOR
%   B13:4/2  MT2231ASC  "BOMBA REFRIG BROCA 1 SOBRECARGA" %
%   B13:4/0  MT2231AFCF  "BOMBA AGUA REFRIG BROCA 1 FALHA CONTATOR FECHAMENTO" %
%   B13:4/3  MT2231SDAT  "BOMBA AGUA REFRIG BROCA 1 DISJUNTOR EM TRIP" %
%   B3:3/1  "BOMBA AGUA REFRIG BROCA 1 DEFEITO" %
% Rung: 2 %
SOR XIC I:9.2/13 OTU B3:3/1 EOR
%   I:9.2/13  P1RESET  "1B10MC2211 BOTAO REARME PERFURATRIZ" %
%   B3:3/1  "BOMBA AGUA REFRIG BROCA 1 DEFEITO" %
% Rung: 3 %
% LIGA BOMBA %
SOR XIC B11:4/0 BST XIC O:9.4/8 XIO I:9.1/5 NXB XIC I:9.1/5 BST XIC I:9.0/1 NXB XIC B11:4/6 BND XIO I:9.0/2 BND OTE O:5.0/8 EOR
%   B11:4/0  MT2231LPP  "BOMBA AGUA REFRIG BROCA 1 PRONTO P PARTIR" %
%   O:9.4/8  VS2238CLAC  "VS2238 VALV DIRECIONAL DE AGUA RESF BROCA ABRIR" %
%   I:9.1/5  C1UHSLOC  "1B3MC2211 UNIDADE HID CHAVE SELETORA LOCAL (MESA DE COMANDO)" %
%   I:9.0/1  MT2231BLIL  "MT2231 MOTOR BOMBA AGUA REFRIG DAS BROCAS BOTAO LIGA" %
%   B11:4/6  MT2231LLI  "BOMBA AGUA REFRIG BROCAS LIGADO" %
%   I:9.0/2  MT2231BDLL  "MT2231 MOTOR BOMBA AGUA REFRIG DAS BROCAS BOTAO DESLIGA" %
%   O:5.0/8  MT2231CLIC  "MOTOR BOMBA AGUA REFRIG BROCAS LIGAR" %

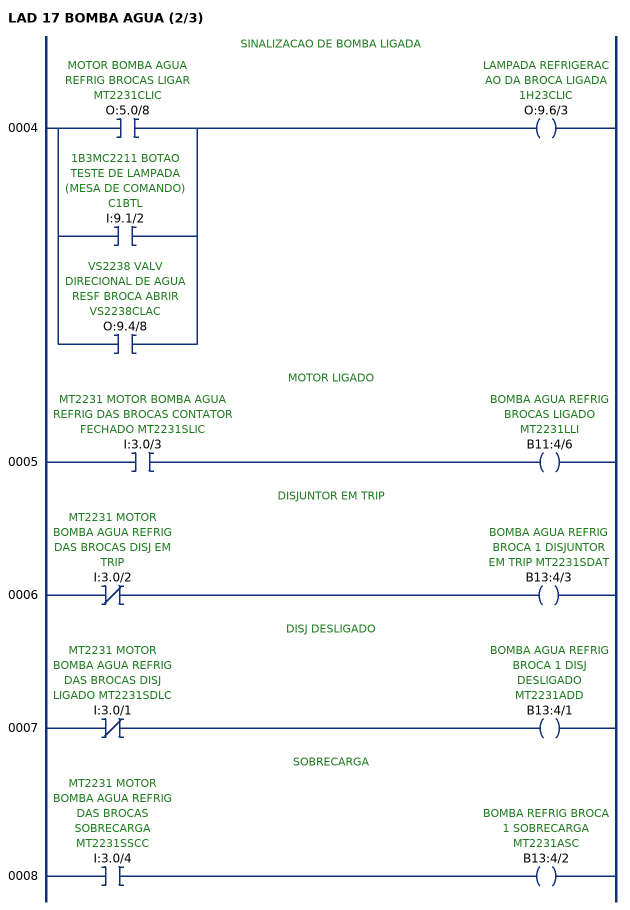
% Rung: 4 %
% SINALIZACAO DE BOMBA LIGADA %
SOR BST XIC O:5.0/8 NXB XIC I:9.1/2 NXB XIC O:9.4/8 BND OTE O:9.6/3 EOR
%   O:5.0/8  MT2231CLIC  "MOTOR BOMBA AGUA REFRIG BROCAS LIGAR" %
%   I:9.1/2  C1BTL  "1B3MC2211 BOTAO TESTE DE LAMPADA (MESA DE COMANDO)" %
%   O:9.4/8  VS2238CLAC  "VS2238 VALV DIRECIONAL DE AGUA RESF BROCA ABRIR" %
%   O:9.6/3  1H23CLIC  "LAMPADA REFRIGERACAO DA BROCA LIGADA" %
% Rung: 5 %
% MOTOR LIGADO %
SOR XIC I:3.0/3 OTE B11:4/6 EOR
%   I:3.0/3  MT2231SLIC  "MT2231 MOTOR BOMBA AGUA REFRIG DAS BROCAS CONTATOR FECHADO" %
%   B11:4/6  MT2231LLI  "BOMBA AGUA REFRIG BROCAS LIGADO" %
% Rung: 6 %
% DISJUNTOR EM TRIP %
SOR XIO I:3.0/2 OTE B13:4/3 EOR
%   I:3.0/2  "MT2231 MOTOR BOMBA AGUA REFRIG DAS BROCAS DISJ EM TRIP" %
%   B13:4/3  MT2231SDAT  "BOMBA AGUA REFRIG BROCA 1 DISJUNTOR EM TRIP" %
% Rung: 7 %
% DISJ DESLIGADO %
SOR XIO I:3.0/1 OTE B13:4/1 EOR
%   I:3.0/1  MT2231SDLC  "MT2231 MOTOR BOMBA AGUA REFRIG DAS BROCAS DISJ LIGADO" %
%   B13:4/1  MT2231ADD  "BOMBA AGUA REFRIG BROCA 1 DISJ DESLIGADO" %
% Rung: 8 %
% SOBRECARGA %
SOR XIC I:3.0/4 OTE B13:4/2 EOR
%   I:3.0/4  MT2231SSCC  "MT2231 MOTOR BOMBA AGUA REFRIG DAS BROCAS SOBRECARGA" %
%   B13:4/2  MT2231ASC  "BOMBA REFRIG BROCA 1 SOBRECARGA" %

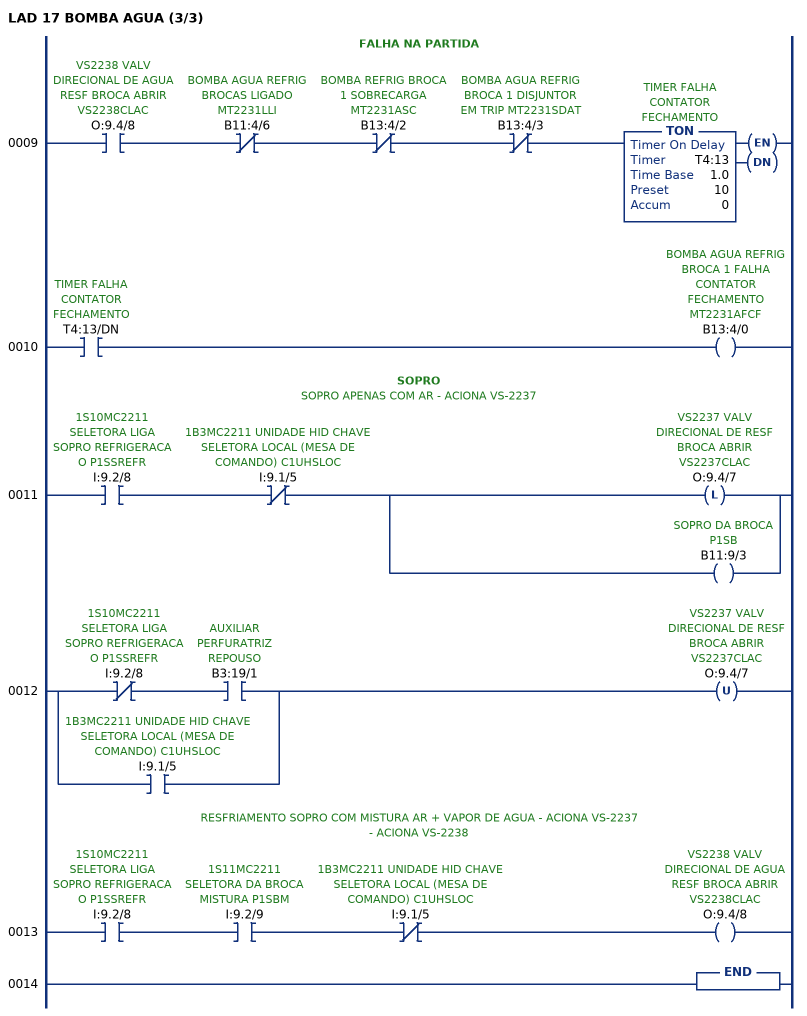
% Rung: 9 %
% TITLE: FALHA NA PARTIDA %
SOR XIC O:9.4/8 XIO B11:4/6 XIO B13:4/2 XIO B13:4/3 TON T4:13 1.0 10 0 EOR
%   O:9.4/8  VS2238CLAC  "VS2238 VALV DIRECIONAL DE AGUA RESF BROCA ABRIR" %
%   B11:4/6  MT2231LLI  "BOMBA AGUA REFRIG BROCAS LIGADO" %
%   B13:4/2  MT2231ASC  "BOMBA REFRIG BROCA 1 SOBRECARGA" %
%   B13:4/3  MT2231SDAT  "BOMBA AGUA REFRIG BROCA 1 DISJUNTOR EM TRIP" %
%   T4:13  "TIMER FALHA CONTATOR FECHAMENTO" %
% Rung: 10 %
SOR XIC T4:13/DN OTE B13:4/0 EOR
%   T4:13  "TIMER FALHA CONTATOR FECHAMENTO" %
%   B13:4/0  MT2231AFCF  "BOMBA AGUA REFRIG BROCA 1 FALHA CONTATOR FECHAMENTO" %
% Rung: 11 %
% TITLE: SOPRO %
% SOPRO APENAS COM AR - ACIONA VS-2237 %
SOR XIC I:9.2/8 XIO I:9.1/5 BST OTL O:9.4/7 NXB OTE B11:9/3 BND EOR
%   I:9.2/8  P1SSREFR  "1S10MC2211 SELETORA LIGA SOPRO REFRIGERACAO" %
%   I:9.1/5  C1UHSLOC  "1B3MC2211 UNIDADE HID CHAVE SELETORA LOCAL (MESA DE COMANDO)" %
%   O:9.4/7  VS2237CLAC  "VS2237 VALV DIRECIONAL DE RESF BROCA ABRIR" %
%   B11:9/3  P1SB  "SOPRO DA BROCA" %
% Rung: 12 %
SOR BST XIO I:9.2/8 XIC B3:19/1 NXB XIC I:9.1/5 BND OTU O:9.4/7 EOR
%   I:9.2/8  P1SSREFR  "1S10MC2211 SELETORA LIGA SOPRO REFRIGERACAO" %
%   B3:19/1  "AUXILIAR PERFURATRIZ REPOUSO" %
%   I:9.1/5  C1UHSLOC  "1B3MC2211 UNIDADE HID CHAVE SELETORA LOCAL (MESA DE COMANDO)" %
%   O:9.4/7  VS2237CLAC  "VS2237 VALV DIRECIONAL DE RESF BROCA ABRIR" %
% Rung: 13 %
% RESFRIAMENTO SOPRO COM MISTURA AR + VAPOR DE AGUA - ACIONA VS-2237
%                                                                                                                                           - ACIONA VS-2238 %
SOR XIC I:9.2/8 XIC I:9.2/9 XIO I:9.1/5 OTE O:9.4/8 EOR
%   I:9.2/8  P1SSREFR  "1S10MC2211 SELETORA LIGA SOPRO REFRIGERACAO" %
%   I:9.2/9  P1SBM  "1S11MC2211 SELETORA DA BROCA MISTURA" %
%   I:9.1/5  C1UHSLOC  "1B3MC2211 UNIDADE HID CHAVE SELETORA LOCAL (MESA DE COMANDO)" %
%   O:9.4/8  VS2238CLAC  "VS2238 VALV DIRECIONAL DE AGUA RESF BROCA ABRIR" %
% Rung: 14 %
SOR END EOR

LADDER 18 "ALR GERAIS"    % ALARMES GERAIS E ANUNCIADOR %
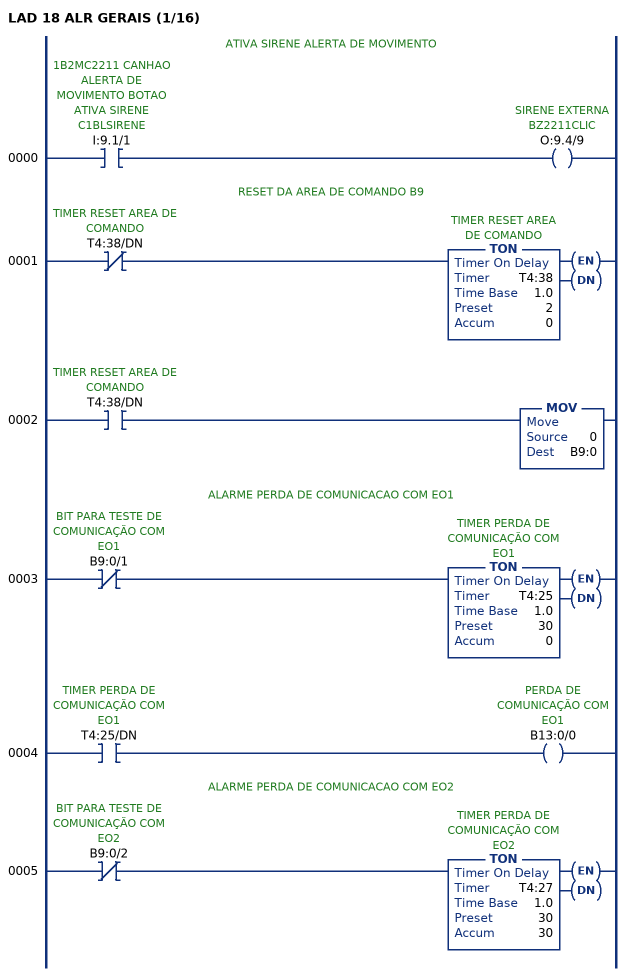
% Rung: 0 %
% ATIVA SIRENE ALERTA DE MOVIMENTO %
SOR XIC I:9.1/1 OTE O:9.4/9 EOR
%   I:9.1/1  C1BLSIRENE  "1B2MC2211 CANHAO ALERTA DE MOVIMENTO BOTAO ATIVA SIRENE" %
%   O:9.4/9  BZ2211CLIC  "SIRENE EXTERNA" %
% Rung: 1 %
% RESET DA AREA DE COMANDO B9 %
SOR XIO T4:38/DN TON T4:38 1.0 2 0 EOR
%   T4:38  "TIMER RESET AREA DE COMANDO" %
% Rung: 2 %
SOR XIC T4:38/DN MOV 0 B9:0 EOR
%   T4:38  "TIMER RESET AREA DE COMANDO" %
% Rung: 3 %
% ALARME PERDA DE COMUNICACAO COM EO1 %
SOR XIO B9:0/1 TON T4:25 1.0 30 0 EOR
%   B9:0/1  "BIT PARA TESTE DE COMUNICAÇÃO COM EO1" %
%   T4:25  "TIMER PERDA DE COMUNICAÇÃO COM EO1" %
% Rung: 4 %
SOR XIC T4:25/DN OTE B13:0/0 EOR
%   T4:25  "TIMER PERDA DE COMUNICAÇÃO COM EO1" %
%   B13:0/0  "PERDA DE COMUNICAÇÃO COM EO1" %
% Rung: 5 %
% ALARME PERDA DE COMUNICACAO COM EO2 %
SOR XIO B9:0/2 TON T4:27 1.0 30 30 EOR
%   B9:0/2  "BIT PARA TESTE DE COMUNICAÇÃO COM EO2" %
%   T4:27  "TIMER PERDA DE COMUNICAÇÃO COM EO2" %

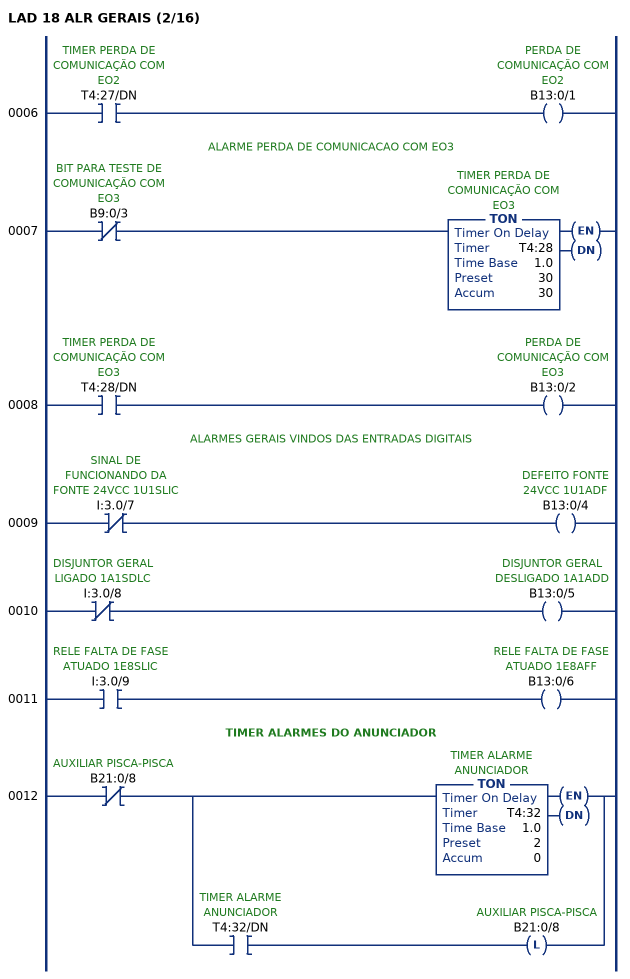
% Rung: 6 %
SOR XIC T4:27/DN OTE B13:0/1 EOR
%   T4:27  "TIMER PERDA DE COMUNICAÇÃO COM EO2" %
%   B13:0/1  "PERDA DE COMUNICAÇÃO COM EO2" %
% Rung: 7 %
% ALARME PERDA DE COMUNICACAO COM EO3 %
SOR XIO B9:0/3 TON T4:28 1.0 30 30 EOR
%   B9:0/3  "BIT PARA TESTE DE COMUNICAÇÃO COM EO3" %
%   T4:28  "TIMER PERDA DE COMUNICAÇÃO COM EO3" %
% Rung: 8 %
SOR XIC T4:28/DN OTE B13:0/2 EOR
%   T4:28  "TIMER PERDA DE COMUNICAÇÃO COM EO3" %
%   B13:0/2  "PERDA DE COMUNICAÇÃO COM EO3" %
% Rung: 9 %
% ALARMES GERAIS VINDOS DAS ENTRADAS DIGITAIS %
SOR XIO I:3.0/7 OTE B13:0/4 EOR
%   I:3.0/7  1U1SLIC  "SINAL DE FUNCIONANDO DA FONTE 24VCC" %
%   B13:0/4  1U1ADF  "DEFEITO FONTE 24VCC" %
% Rung: 10 %
SOR XIO I:3.0/8 OTE B13:0/5 EOR
%   I:3.0/8  1A1SDLC  "DISJUNTOR GERAL LIGADO" %
%   B13:0/5  1A1ADD  "DISJUNTOR GERAL DESLIGADO" %
% Rung: 11 %
SOR XIC I:3.0/9 OTE B13:0/6 EOR
%   I:3.0/9  1E8SLIC  "RELE FALTA DE FASE ATUADO" %
%   B13:0/6  1E8AFF  "RELE FALTA DE FASE ATUADO" %
% Rung: 12 %
% TITLE: TIMER ALARMES DO ANUNCIADOR %
SOR XIO B21:0/8 BST TON T4:32 1.0 2 0 NXB XIC T4:32/DN OTL B21:0/8 BND EOR
%   B21:0/8  "AUXILIAR PISCA-PISCA" %
%   T4:32  "TIMER ALARME ANUNCIADOR" %

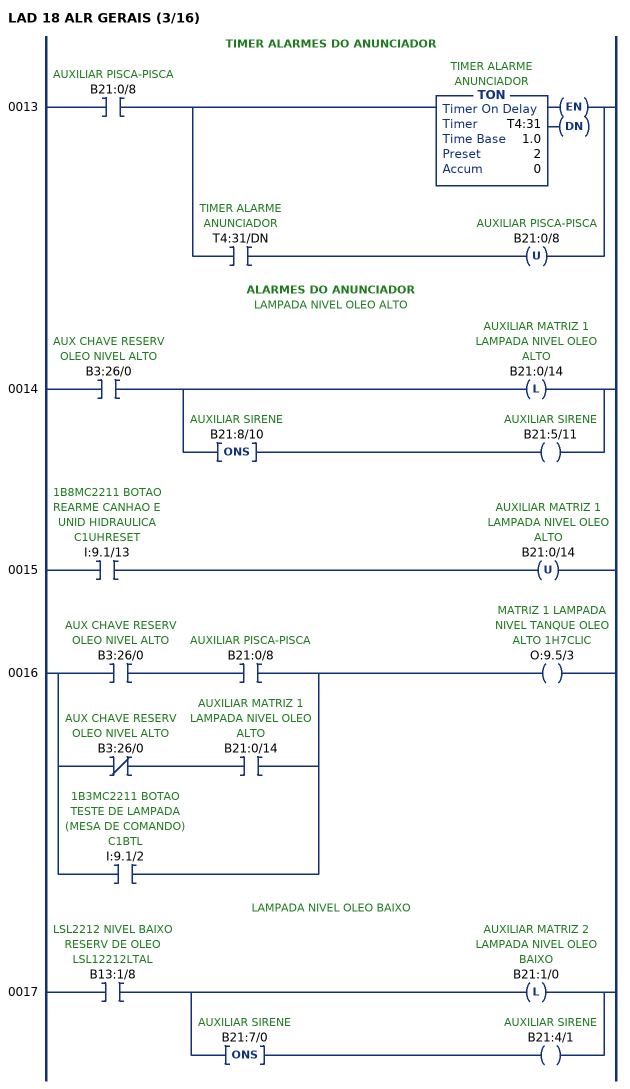
% Rung: 13 %
% TITLE: TIMER ALARMES DO ANUNCIADOR %
SOR XIC B21:0/8 BST TON T4:31 1.0 2 0 NXB XIC T4:31/DN OTU B21:0/8 BND EOR
%   B21:0/8  "AUXILIAR PISCA-PISCA" %
%   T4:31  "TIMER ALARME ANUNCIADOR" %
% Rung: 14 %
% TITLE: ALARMES DO ANUNCIADOR %
% LAMPADA NIVEL OLEO ALTO %
SOR XIC B3:26/0 BST OTL B21:0/14 NXB OSR B21:8/10 OTE B21:5/11 BND EOR
%   B3:26/0  "AUX CHAVE RESERV OLEO NIVEL ALTO" %
%   B21:0/14  "AUXILIAR MATRIZ 1 LAMPADA NIVEL OLEO ALTO" %
%   B21:8/10  "AUXILIAR SIRENE" %
%   B21:5/11  "AUXILIAR SIRENE" %
% Rung: 15 %
SOR XIC I:9.1/13 OTU B21:0/14 EOR
%   I:9.1/13  C1UHRESET  "1B8MC2211 BOTAO REARME CANHAO E UNID HIDRAULICA" %
%   B21:0/14  "AUXILIAR MATRIZ 1 LAMPADA NIVEL OLEO ALTO" %
% Rung: 16 %
SOR BST XIC B3:26/0 XIC B21:0/8 NXB XIO B3:26/0 XIC B21:0/14 NXB XIC I:9.1/2 BND OTE O:9.5/3 EOR
%   B3:26/0  "AUX CHAVE RESERV OLEO NIVEL ALTO" %
%   B21:0/8  "AUXILIAR PISCA-PISCA" %
%   B21:0/14  "AUXILIAR MATRIZ 1 LAMPADA NIVEL OLEO ALTO" %
%   I:9.1/2  C1BTL  "1B3MC2211 BOTAO TESTE DE LAMPADA (MESA DE COMANDO)" %
%   O:9.5/3  1H7CLIC  "MATRIZ 1 LAMPADA NIVEL TANQUE OLEO ALTO" %
% Rung: 17 %
% LAMPADA NIVEL OLEO BAIXO %
SOR XIC B13:1/8 BST OTL B21:1/0 NXB OSR B21:7/0 OTE B21:4/1 BND EOR
%   B13:1/8  LSL12212LTAL  "LSL2212 NIVEL BAIXO RESERV DE OLEO" %
%   B21:1/0  "AUXILIAR MATRIZ 2 LAMPADA NIVEL OLEO BAIXO" %
%   B21:7/0  "AUXILIAR SIRENE" %
%   B21:4/1  "AUXILIAR SIRENE" %

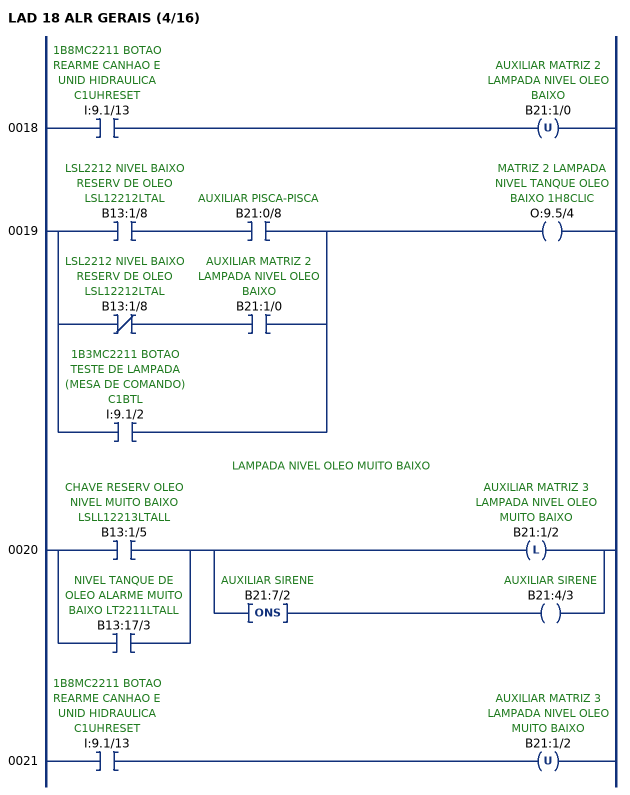
% Rung: 18 %
SOR XIC I:9.1/13 OTU B21:1/0 EOR
%   I:9.1/13  C1UHRESET  "1B8MC2211 BOTAO REARME CANHAO E UNID HIDRAULICA" %
%   B21:1/0  "AUXILIAR MATRIZ 2 LAMPADA NIVEL OLEO BAIXO" %
% Rung: 19 %
SOR BST XIC B13:1/8 XIC B21:0/8 NXB XIO B13:1/8 XIC B21:1/0 NXB XIC I:9.1/2 BND OTE O:9.5/4 EOR
%   B13:1/8  LSL12212LTAL  "LSL2212 NIVEL BAIXO RESERV DE OLEO" %
%   B21:0/8  "AUXILIAR PISCA-PISCA" %
%   B21:1/0  "AUXILIAR MATRIZ 2 LAMPADA NIVEL OLEO BAIXO" %
%   I:9.1/2  C1BTL  "1B3MC2211 BOTAO TESTE DE LAMPADA (MESA DE COMANDO)" %
%   O:9.5/4  1H8CLIC  "MATRIZ 2 LAMPADA NIVEL TANQUE OLEO BAIXO" %
% Rung: 20 %
% LAMPADA NIVEL OLEO MUITO BAIXO %
SOR BST XIC B13:1/5 NXB XIC B13:17/3 BND BST OTL B21:1/2 NXB OSR B21:7/2 OTE B21:4/3 BND EOR
%   B13:1/5  LSLL12213LTALL  "CHAVE RESERV OLEO NIVEL MUITO BAIXO" %
%   B13:17/3  LT2211LTALL  "NIVEL TANQUE DE OLEO ALARME MUITO BAIXO" %
%   B21:1/2  "AUXILIAR MATRIZ 3 LAMPADA NIVEL OLEO MUITO BAIXO" %
%   B21:7/2  "AUXILIAR SIRENE" %
%   B21:4/3  "AUXILIAR SIRENE" %
% Rung: 21 %
SOR XIC I:9.1/13 OTU B21:1/2 EOR
%   I:9.1/13  C1UHRESET  "1B8MC2211 BOTAO REARME CANHAO E UNID HIDRAULICA" %
%   B21:1/2  "AUXILIAR MATRIZ 3 LAMPADA NIVEL OLEO MUITO BAIXO" %

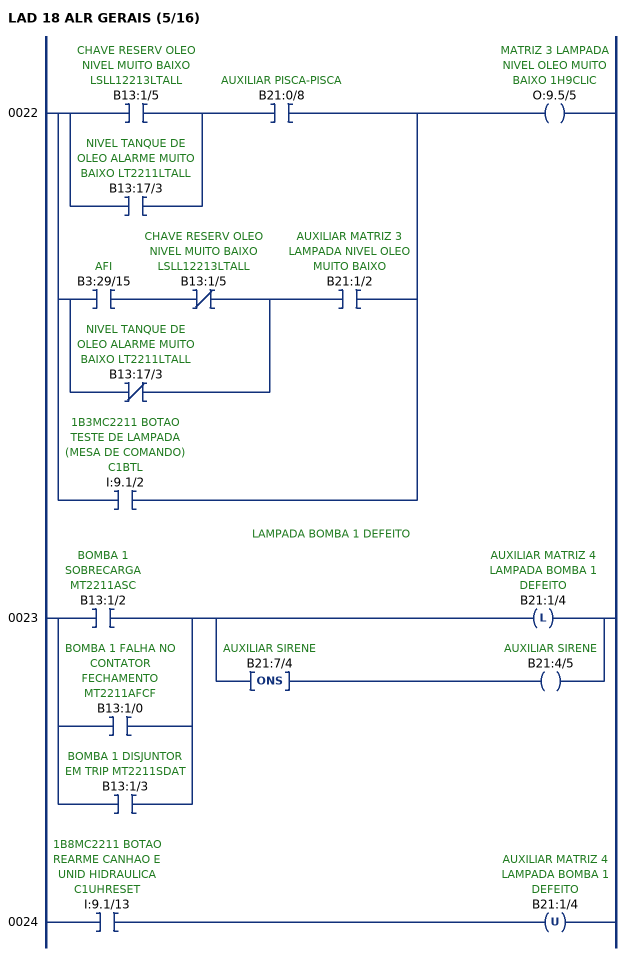
% Rung: 22 %
SOR BST BST XIC B13:1/5 NXB XIC B13:17/3 BND XIC B21:0/8 NXB BST XIC B3:29/15 XIO B13:1/5 NXB XIO B13:17/3 BND XIC B21:1/2 NXB XIC I:9.1/2 BND OTE O:9.5/5 EOR
%   B13:1/5  LSLL12213LTALL  "CHAVE RESERV OLEO NIVEL MUITO BAIXO" %
%   B13:17/3  LT2211LTALL  "NIVEL TANQUE DE OLEO ALARME MUITO BAIXO" %
%   B21:0/8  "AUXILIAR PISCA-PISCA" %
%   B3:29/15  AFI %
%   B21:1/2  "AUXILIAR MATRIZ 3 LAMPADA NIVEL OLEO MUITO BAIXO" %
%   I:9.1/2  C1BTL  "1B3MC2211 BOTAO TESTE DE LAMPADA (MESA DE COMANDO)" %
%   O:9.5/5  1H9CLIC  "MATRIZ 3 LAMPADA NIVEL OLEO MUITO BAIXO" %
% Rung: 23 %
% LAMPADA BOMBA 1 DEFEITO %
SOR BST XIC B13:1/2 NXB XIC B13:1/0 NXB XIC B13:1/3 BND BST OTL B21:1/4 NXB OSR B21:7/4 OTE B21:4/5 BND EOR
%   B13:1/2  MT2211ASC  "BOMBA 1 SOBRECARGA" %
%   B13:1/0  MT2211AFCF  "BOMBA 1 FALHA NO CONTATOR FECHAMENTO" %
%   B13:1/3  MT2211SDAT  "BOMBA 1 DISJUNTOR EM TRIP" %
%   B21:1/4  "AUXILIAR MATRIZ 4 LAMPADA BOMBA 1 DEFEITO" %
%   B21:7/4  "AUXILIAR SIRENE" %
%   B21:4/5  "AUXILIAR SIRENE" %
% Rung: 24 %
SOR XIC I:9.1/13 OTU B21:1/4 EOR
%   I:9.1/13  C1UHRESET  "1B8MC2211 BOTAO REARME CANHAO E UNID HIDRAULICA" %
%   B21:1/4  "AUXILIAR MATRIZ 4 LAMPADA BOMBA 1 DEFEITO" %

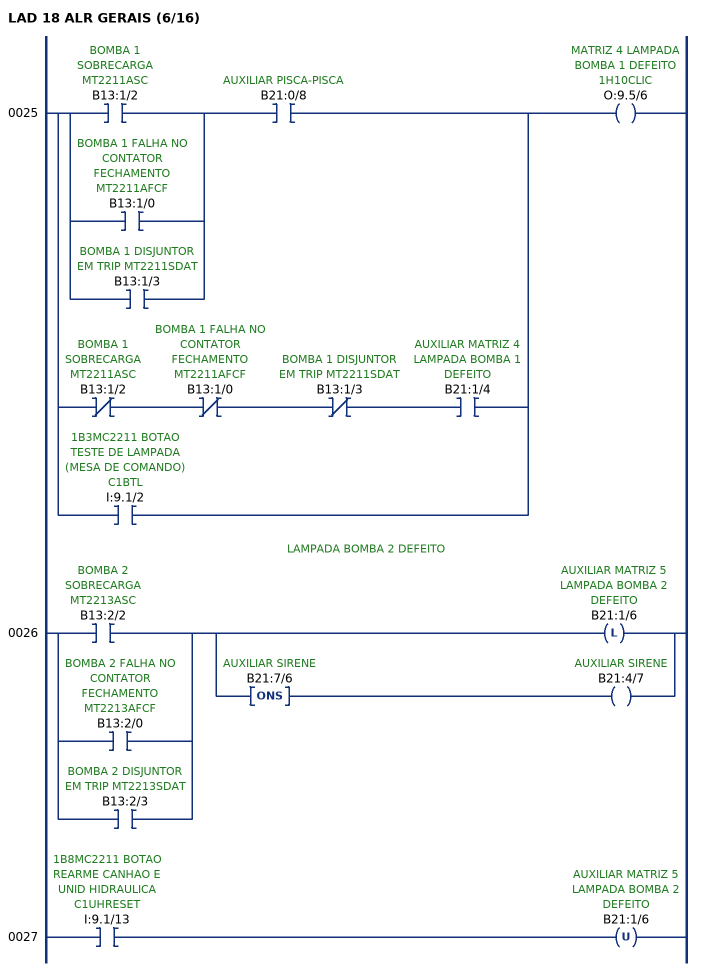
% Rung: 25 %
SOR BST BST XIC B13:1/2 NXB XIC B13:1/0 NXB XIC B13:1/3 BND XIC B21:0/8 NXB XIO B13:1/2 XIO B13:1/0 XIO B13:1/3 XIC B21:1/4 NXB XIC I:9.1/2 BND OTE O:9.5/6 EOR
%   B13:1/2  MT2211ASC  "BOMBA 1 SOBRECARGA" %
%   B13:1/0  MT2211AFCF  "BOMBA 1 FALHA NO CONTATOR FECHAMENTO" %
%   B13:1/3  MT2211SDAT  "BOMBA 1 DISJUNTOR EM TRIP" %
%   B21:0/8  "AUXILIAR PISCA-PISCA" %
%   B21:1/4  "AUXILIAR MATRIZ 4 LAMPADA BOMBA 1 DEFEITO" %
%   I:9.1/2  C1BTL  "1B3MC2211 BOTAO TESTE DE LAMPADA (MESA DE COMANDO)" %
%   O:9.5/6  1H10CLIC  "MATRIZ 4 LAMPADA BOMBA 1 DEFEITO" %
% Rung: 26 %
% LAMPADA BOMBA 2 DEFEITO %
SOR BST XIC B13:2/2 NXB XIC B13:2/0 NXB XIC B13:2/3 BND BST OTL B21:1/6 NXB OSR B21:7/6 OTE B21:4/7 BND EOR
%   B13:2/2  MT2213ASC  "BOMBA 2 SOBRECARGA" %
%   B13:2/0  MT2213AFCF  "BOMBA 2 FALHA NO CONTATOR FECHAMENTO" %
%   B13:2/3  MT2213SDAT  "BOMBA 2 DISJUNTOR EM TRIP" %
%   B21:1/6  "AUXILIAR MATRIZ 5 LAMPADA BOMBA 2 DEFEITO" %
%   B21:7/6  "AUXILIAR SIRENE" %
%   B21:4/7  "AUXILIAR SIRENE" %
% Rung: 27 %
SOR XIC I:9.1/13 OTU B21:1/6 EOR
%   I:9.1/13  C1UHRESET  "1B8MC2211 BOTAO REARME CANHAO E UNID HIDRAULICA" %
%   B21:1/6  "AUXILIAR MATRIZ 5 LAMPADA BOMBA 2 DEFEITO" %

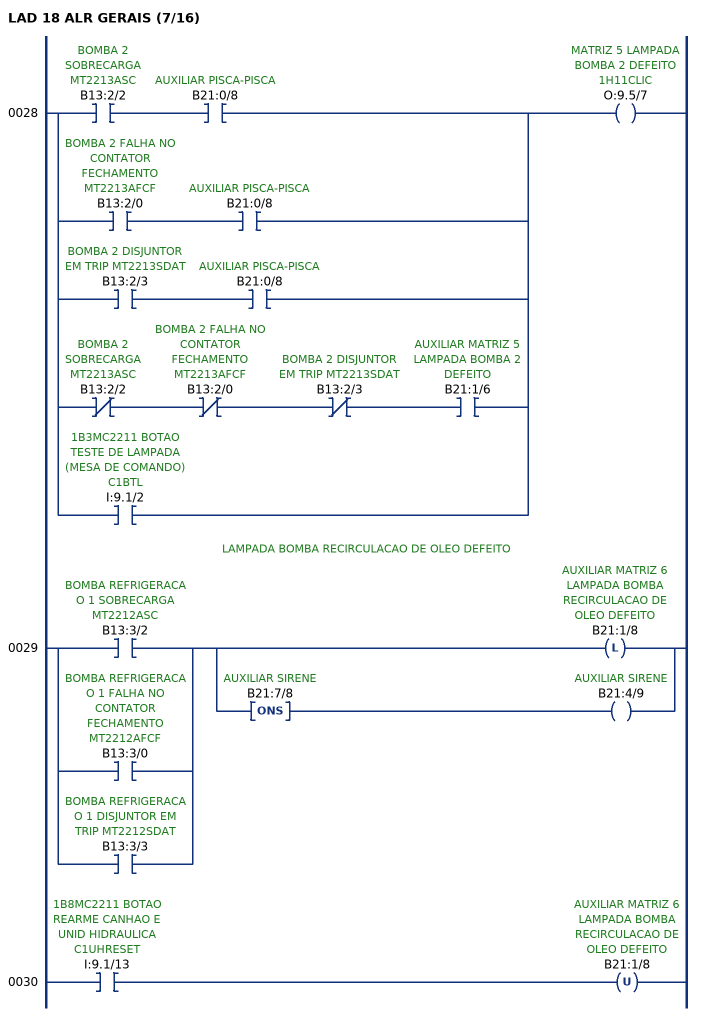
% Rung: 28 %
SOR BST BST XIC B13:2/2 XIC B21:0/8 NXB XIC B13:2/0 XIC B21:0/8 NXB XIC B13:2/3 XIC B21:0/8 BND NXB XIO B13:2/2 XIO B13:2/0 XIO B13:2/3 XIC B21:1/6 NXB XIC I:9.1/2 BND OTE O:9.5/7 EOR
%   B13:2/2  MT2213ASC  "BOMBA 2 SOBRECARGA" %
%   B21:0/8  "AUXILIAR PISCA-PISCA" %
%   B13:2/0  MT2213AFCF  "BOMBA 2 FALHA NO CONTATOR FECHAMENTO" %
%   B13:2/3  MT2213SDAT  "BOMBA 2 DISJUNTOR EM TRIP" %
%   B21:1/6  "AUXILIAR MATRIZ 5 LAMPADA BOMBA 2 DEFEITO" %
%   I:9.1/2  C1BTL  "1B3MC2211 BOTAO TESTE DE LAMPADA (MESA DE COMANDO)" %
%   O:9.5/7  1H11CLIC  "MATRIZ 5 LAMPADA BOMBA 2 DEFEITO" %
% Rung: 29 %
% LAMPADA BOMBA RECIRCULACAO DE OLEO DEFEITO %
SOR BST XIC B13:3/2 NXB XIC B13:3/0 NXB XIC B13:3/3 BND BST OTL B21:1/8 NXB OSR B21:7/8 OTE B21:4/9 BND EOR
%   B13:3/2  MT2212ASC  "BOMBA REFRIGERACAO 1 SOBRECARGA" %
%   B13:3/0  MT2212AFCF  "BOMBA REFRIGERACAO 1 FALHA NO CONTATOR FECHAMENTO" %
%   B13:3/3  MT2212SDAT  "BOMBA REFRIGERACAO 1 DISJUNTOR EM TRIP" %
%   B21:1/8  "AUXILIAR MATRIZ 6 LAMPADA BOMBA RECIRCULACAO DE OLEO DEFEITO" %
%   B21:7/8  "AUXILIAR SIRENE" %
%   B21:4/9  "AUXILIAR SIRENE" %
% Rung: 30 %
SOR XIC I:9.1/13 OTU B21:1/8 EOR
%   I:9.1/13  C1UHRESET  "1B8MC2211 BOTAO REARME CANHAO E UNID HIDRAULICA" %
%   B21:1/8  "AUXILIAR MATRIZ 6 LAMPADA BOMBA RECIRCULACAO DE OLEO DEFEITO" %

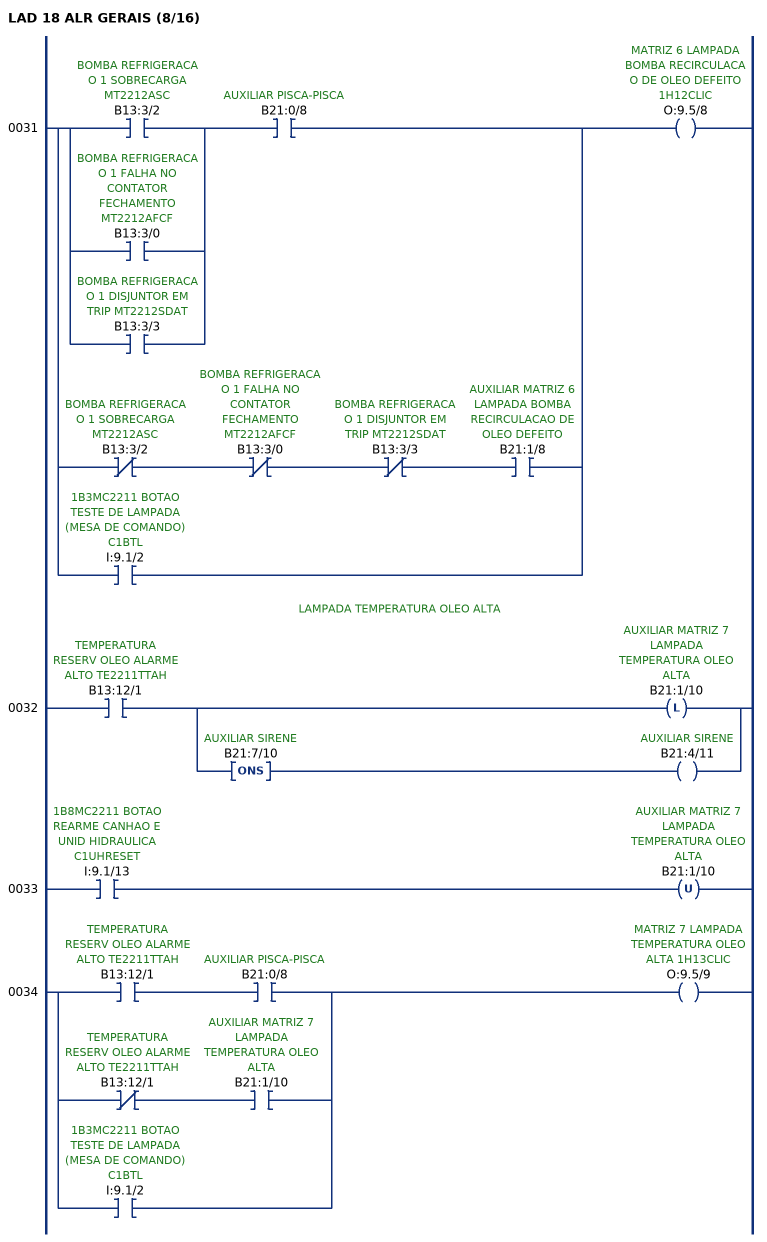
% Rung: 31 %
SOR BST BST XIC B13:3/2 NXB XIC B13:3/0 NXB XIC B13:3/3 BND XIC B21:0/8 NXB XIO B13:3/2 XIO B13:3/0 XIO B13:3/3 XIC B21:1/8 NXB XIC I:9.1/2 BND OTE O:9.5/8 EOR
%   B13:3/2  MT2212ASC  "BOMBA REFRIGERACAO 1 SOBRECARGA" %
%   B13:3/0  MT2212AFCF  "BOMBA REFRIGERACAO 1 FALHA NO CONTATOR FECHAMENTO" %
%   B13:3/3  MT2212SDAT  "BOMBA REFRIGERACAO 1 DISJUNTOR EM TRIP" %
%   B21:0/8  "AUXILIAR PISCA-PISCA" %
%   B21:1/8  "AUXILIAR MATRIZ 6 LAMPADA BOMBA RECIRCULACAO DE OLEO DEFEITO" %
%   I:9.1/2  C1BTL  "1B3MC2211 BOTAO TESTE DE LAMPADA (MESA DE COMANDO)" %
%   O:9.5/8  1H12CLIC  "MATRIZ 6 LAMPADA BOMBA RECIRCULACAO DE OLEO DEFEITO" %
% Rung: 32 %
% LAMPADA TEMPERATURA OLEO ALTA %
SOR XIC B13:12/1 BST OTL B21:1/10 NXB OSR B21:7/10 OTE B21:4/11 BND EOR
%   B13:12/1  TE2211TTAH  "TEMPERATURA RESERV OLEO ALARME ALTO" %
%   B21:1/10  "AUXILIAR MATRIZ 7 LAMPADA TEMPERATURA OLEO ALTA" %
%   B21:7/10  "AUXILIAR SIRENE" %
%   B21:4/11  "AUXILIAR SIRENE" %
% Rung: 33 %
SOR XIC I:9.1/13 OTU B21:1/10 EOR
%   I:9.1/13  C1UHRESET  "1B8MC2211 BOTAO REARME CANHAO E UNID HIDRAULICA" %
%   B21:1/10  "AUXILIAR MATRIZ 7 LAMPADA TEMPERATURA OLEO ALTA" %
% Rung: 34 %
SOR BST XIC B13:12/1 XIC B21:0/8 NXB XIO B13:12/1 XIC B21:1/10 NXB XIC I:9.1/2 BND OTE O:9.5/9 EOR
%   B13:12/1  TE2211TTAH  "TEMPERATURA RESERV OLEO ALARME ALTO" %
%   B21:0/8  "AUXILIAR PISCA-PISCA" %
%   B21:1/10  "AUXILIAR MATRIZ 7 LAMPADA TEMPERATURA OLEO ALTA" %
%   I:9.1/2  C1BTL  "1B3MC2211 BOTAO TESTE DE LAMPADA (MESA DE COMANDO)" %
%   O:9.5/9  1H13CLIC  "MATRIZ 7 LAMPADA TEMPERATURA OLEO ALTA" %

